C09087=1078.769,309.066,-90.171,175.453,27.389,154.727
C09088=1078.775,309.314,-90.203,175.457,27.393,154.728
C09089=1078.781,309.562,-90.235,175.459,27.397,154.729
C09090=1078.787,309.810,-90.267,175.462,27.402,154.729
C09091=1078.793,310.058,-90.299,175.465,27.406,154.730
C09092=1078.799,310.305,-90.330,175.468,27.410,154.730
C09093=1078.805,310.553,-90.362,175.471,27.415,154.731
C09094=1078.811,310.801,-90.394,175.474,27.419,154.732
C09095=1078.817,311.049,-90.426,175.477,27.423,154.733
C09096=1078.823,311.297,-90.458,175.480,27.427,154.733
C09097=1078.829,311.545,-90.490,175.483,27.432,154.734
C09098=1078.835,311.793,-90.522,175.486,27.436,154.735
C09099=1078.841,312.040,-90.553,175.489,27.440,154.735
C09100=1078.847,312.289,-90.585,175.492,27.444,154.736
C09101=1078.853,312.536,-90.618,175.495,27.448,154.736
C09102=1078.859,312.783,-90.649,175.497,27.452,154.737
C09103=1078.865,313.032,-90.681,175.501,27.457,154.738
C09104=1078.871,313.280,-90.713,175.504,27.461,154.738
C09105=1078.877,313.527,-90.746,175.507,27.465,154.739
C09106=1078.883,313.776,-90.778,175.510,27.469,154.740
C09107=1078.889,314.023,-90.810,175.512,27.474,154.740
C09108=1078.895,314.271,-90.841,175.515,27.478,154.741
C09109=1078.902,314.519,-90.874,175.519,27.482,154.742
C09110=1078.908,314.767,-90.906,175.522,27.487,154.742
C09111=1078.914,315.015,-90.938,175.525,27.491,154.743
C09112=1078.919,315.262,-90.971,175.527,27.495,154.744
C09113=1078.925,315.511,-91.003,175.530,27.500,154.745
C09114=1078.931,315.758,-91.036,175.534,27.504,154.745
C09115=1078.936,316.006,-91.067,175.537,27.509,154.746
C09116=1078.942,316.254,-91.101,175.539,27.513,154.747
C09117=1078.947,316.467,-91.129,175.542,27.517,154.747
C09118=1078.952,316.679,-91.156,175.544,27.521,154.748
C09119=1078.957,316.892,-91.184,175.547,27.524,154.748
C09120=1078.962,317.104,-91.212,175.550,27.528,154.749
C09121=1078.967,317.317,-91.240,175.552,27.532,154.750
C09122=1078.972,317.530,-91.268,175.555,27.536,154.750
C09123=1078.977,317.742,-91.295,175.557,27.540,154.751
C09124=1078.982,317.955,-91.323,175.560,27.543,154.751
C09125=1078.988,318.203,-91.355,175.562,27.548,154.752
C09126=1078.993,318.451,-91.388,175.566,27.552,154.753
C09127=1078.999,318.699,-91.420,175.569,27.557,154.754
C09128=1079.005,318.946,-91.453,175.572,27.561,154.754
C09129=1079.011,319.194,-91.486,175.575,27.566,154.755
C09130=1079.017,319.443,-91.518,175.578,27.570,154.756
C09131=1079.023,319.690,-91.551,175.580,27.575,154.757
C09132=1079.028,319.937,-91.584,175.583,27.579,154.757
C09133=1079.034,320.186,-91.616,175.587,27.584,154.758
C09134=1079.041,320.433,-91.649,175.590,27.588,154.759
C09135=1079.046,320.681,-91.682,175.593,27.593,154.759
C09136=1079.052,320.929,-91.715,175.596,27.597,154.760
C09137=1079.058,321.177,-91.747,175.598,27.601,154.761
C09138=1079.064,321.425,-91.780,175.602,27.606,154.762
C09139=1079.070,321.672,-91.813,175.605,27.611,154.762
C09140=1079.077,321.920,-91.846,175.608,27.615,154.763
C09141=1079.082,322.168,-91.879,175.611,27.620,154.764
C09142=1079.087,322.415,-91.911,175.614,27.624,154.764
C09143=1079.093,322.663,-91.944,175.617,27.629,154.765
C09144=1079.099,322.911,-91.977,175.619,27.633,154.766
C09145=1079.106,323.158,-92.010,175.623,27.637,154.767
C09146=1079.111,323.406,-92.043,175.626,27.642,154.767
C09147=1079.117,323.654,-92.076,175.629,27.647,154.768
C09148=1079.123,323.902,-92.109,175.632,27.651,154.769
C09149=1079.129,324.149,-92.142,175.635,27.656,154.770
C09150=1079.135,324.397,-92.175,175.638,27.661,154.770
C09151=1079.141,324.645,-92.208,175.642,27.665,154.771
C09152=1079.147,324.893,-92.241,175.644,27.669,154.772
C09153=1079.153,325.140,-92.274,175.647,27.674,154.773
C09154=1079.160,325.389,-92.307,175.650,27.678,154.773
C09155=1079.165,325.637,-92.340,175.653,27.683,154.774
C09156=1079.172,325.884,-92.373,175.656,27.688,154.775
C09157=1079.177,326.132,-92.407,175.660,27.692,154.775
C09158=1079.184,326.380,-92.439,175.663,27.697,154.776
C09159=1079.189,326.628,-92.473,175.666,27.701,154.777
C09160=1079.195,326.875,-92.505,175.669,27.706,154.778
C09161=1079.201,327.123,-92.539,175.672,27.710,154.778
C09162=1079.208,327.370,-92.572,175.675,27.715,154.779
C09163=1079.213,327.618,-92.605,175.678,27.720,154.780
C09164=1079.220,327.866,-92.639,175.681,27.724,154.781
C09165=1079.226,328.114,-92.672,175.684,27.728,154.781
C09166=1079.232,328.361,-92.705,175.687,27.733,154.782
C09167=1079.238,328.609,-92.739,175.690,27.738,154.783
C09168=1079.244,328.857,-92.771,175.693,27.743,154.784
C09169=1079.250,329.105,-92.805,175.697,27.747,154.785
C09170=1079.257,329.352,-92.839,175.700,27.752,154.785
C09171=1079.262,329.600,-92.872,175.703,27.756,154.786
C09172=1079.269,329.848,-92.905,175.706,27.761,154.787
C09173=1079.279,330.266,-92.961,175.712,27.769,154.788
C09174=1079.289,330.685,-93.018,175.716,27.776,154.789
C09175=1079.300,331.104,-93.075,175.722,27.785,154.791
C09176=1079.310,331.523,-93.131,175.727,27.793,154.792
C09177=1079.316,331.770,-93.165,175.731,27.797,154.793
C09178=1079.322,332.018,-93.199,175.734,27.802,154.793
C09179=1079.328,332.266,-93.232,175.737,27.807,154.794
C09180=1079.334,332.513,-93.266,175.740,27.812,154.795
C09181=1079.340,332.761,-93.299,175.743,27.816,154.796
C09182=1079.346,333.009,-93.333,175.746,27.821,154.797
C09183=1079.352,333.257,-93.367,175.749,27.826,154.797
C09184=1079.358,333.504,-93.401,175.753,27.831,154.798
C09185=1079.364,333.752,-93.435,175.756,27.836,154.799
C09186=1079.369,334.000,-93.468,175.759,27.840,154.800
C09187=1079.376,334.247,-93.502,175.762,27.845,154.801
C09188=1079.382,334.495,-93.536,175.765,27.850,154.801
C09189=1079.388,334.742,-93.570,175.768,27.855,154.802
C09190=1079.394,334.990,-93.604,175.771,27.860,154.803
C09191=1079.400,335.238,-93.638,175.775,27.864,154.804
C09192=1079.406,335.486,-93.671,175.778,27.870,154.805
C09193=1079.411,335.733,-93.706,175.781,27.874,154.805
C09194=1079.418,335.981,-93.740,175.784,27.879,154.806
C09195=1079.424,336.228,-93.774,175.787,27.884,154.807
C09196=1079.430,336.475,-93.808,175.790,27.889,154.808
C09197=1079.436,336.724,-93.842,175.793,27.894,154.809
C09198=1079.442,336.971,-93.876,175.797,27.898,154.809
C09199=1079.448,337.219,-93.910,175.800,27.904,154.810
C09200=1079.455,337.466,-93.944,175.803,27.908,154.811
C09201=1079.461,337.714,-93.978,175.806,27.913,154.812
C09202=1079.467,337.962,-94.012,175.809,27.918,154.813
C09203=1079.473,338.209,-94.046,175.812,27.923,154.814
C09204=1079.478,338.456,-94.081,175.815,27.928,154.815
C09205=1079.484,338.704,-94.115,175.819,27.933,154.815
C09206=1079.490,338.952,-94.149,175.822,27.938,154.816
C09207=1079.496,339.199,-94.183,175.825,27.943,154.817
C09208=1079.503,339.447,-94.218,175.828,27.948,154.818
C09209=1079.509,339.694,-94.252,175.831,27.952,154.819
C09210=1079.515,339.942,-94.286,175.834,27.958,154.820
C09211=1079.520,340.190,-94.321,175.837,27.963,154.820
C09212=1079.526,340.437,-94.355,175.840,27.968,154.821
C09213=1079.532,340.685,-94.389,175.844,27.973,154.822
C09214=1079.538,340.932,-94.423,175.848,27.978,154.823
C09215=1079.545,341.180,-94.458,175.851,27.983,154.824
C09216=1079.551,341.428,-94.492,175.854,27.988,154.825
C09217=1079.556,341.676,-94.527,175.857,27.993,154.825
C09218=1079.563,341.923,-94.562,175.860,27.998,154.826
C09219=1079.569,342.171,-94.596,175.863,28.003,154.827
C09220=1079.575,342.418,-94.630,175.866,28.008,154.828
C09221=1079.581,342.666,-94.665,175.870,28.013,154.829
C09222=1079.587,342.913,-94.700,175.873,28.018,154.830
C09223=1079.593,343.161,-94.734,175.876,28.023,154.831
C09224=1079.599,343.408,-94.768,175.879,28.028,154.832
C09225=1079.609,343.822,-94.827,175.884,28.037,154.833
C09226=1079.619,344.235,-94.884,175.890,28.045,154.834
C09227=1079.630,344.648,-94.942,175.895,28.054,154.836
C09228=1079.640,345.061,-95.000,175.901,28.062,154.837
C09229=1079.646,345.309,-95.035,175.904,28.067,154.838
C09230=1079.651,345.556,-95.070,175.907,28.073,154.839
C09231=1079.658,345.804,-95.105,175.910,28.078,154.840
C09232=1079.664,346.052,-95.140,175.914,28.083,154.841
C09233=1079.670,346.299,-95.174,175.918,28.088,154.842
C09234=1079.676,346.547,-95.210,175.921,28.094,154.843
C09235=1079.682,346.794,-95.244,175.924,28.099,154.844
C09236=1079.688,347.042,-95.279,175.927,28.104,154.845
C09237=1079.694,347.289,-95.315,175.930,28.109,154.846
C09238=1079.700,347.537,-95.349,175.933,28.114,154.846
C09239=1079.706,347.784,-95.385,175.937,28.120,154.847
C09240=1079.712,348.032,-95.419,175.940,28.125,154.848
C09241=1079.718,348.279,-95.455,175.943,28.131,154.849
C09242=1079.725,348.527,-95.490,175.946,28.136,154.850
C09243=1079.730,348.774,-95.525,175.950,28.141,154.851
C09244=1079.737,349.022,-95.559,175.953,28.146,154.852
C09245=1079.743,349.269,-95.595,175.957,28.152,154.853
C09246=1079.748,349.516,-95.631,175.960,28.157,154.854
C09247=1079.755,349.764,-95.666,175.963,28.162,154.855
C09248=1079.761,350.012,-95.701,175.966,28.168,154.856
C09249=1079.767,350.258,-95.735,175.969,28.173,154.857
C09250=1079.773,350.506,-95.771,175.973,28.179,154.858
C09251=1079.780,350.754,-95.806,175.976,28.184,154.859
C09252=1079.785,351.001,-95.842,175.979,28.189,154.859
C09253=1079.791,351.248,-95.877,175.983,28.195,154.860
C09254=1079.798,351.496,-95.912,175.986,28.200,154.861
C09255=1079.804,351.744,-95.948,175.990,28.205,154.862
C09256=1079.810,351.991,-95.982,175.993,28.211,154.863
C09257=1079.816,352.238,-96.018,175.996,28.216,154.864
C09258=1079.822,352.486,-96.054,175.999,28.221,154.865
C09259=1079.829,352.733,-96.089,176.002,28.227,154.866
C09260=1079.834,352.980,-96.124,176.006,28.232,154.867
C09261=1079.840,353.228,-96.160,176.009,28.238,154.868
C09262=1079.847,353.475,-96.195,176.012,28.243,154.869
C09263=1079.853,353.723,-96.231,176.016,28.249,154.870
C09264=1079.859,353.969,-96.267,176.020,28.254,154.871
C09265=1079.865,354.217,-96.303,176.023,28.260,154.872
C09266=1079.871,354.465,-96.338,176.026,28.265,154.873
C09267=1079.878,354.712,-96.374,176.029,28.271,154.874
C09268=1079.884,354.960,-96.409,176.033,28.276,154.875
C09269=1079.889,355.207,-96.445,176.036,28.282,154.876
C09270=1079.895,355.454,-96.481,176.039,28.287,154.877
C09271=1079.901,355.701,-96.517,176.042,28.293,154.878
C09272=1079.907,355.949,-96.553,176.046,28.299,154.879
C09273=1079.914,356.196,-96.588,176.049,28.304,154.880
C09274=1079.921,356.443,-96.624,176.052,28.310,154.881
C09275=1079.926,356.690,-96.660,176.056,28.315,154.882
C09276=1079.932,356.938,-96.695,176.060,28.321,154.883
C09277=1079.941,357.295,-96.747,176.064,28.329,154.884
C09278=1079.950,357.652,-96.799,176.069,28.337,154.886
C09279=1079.959,358.010,-96.851,176.074,28.345,154.887
C09280=1079.968,358.367,-96.903,176.078,28.353,154.889
C09281=1079.974,358.615,-96.939,176.082,28.359,154.890
C09282=1079.981,358.862,-96.975,176.085,28.365,154.891
C09283=1079.987,359.110,-97.011,176.089,28.371,154.892
C09284=1079.993,359.357,-97.047,176.093,28.377,154.893
C09285=1079.999,359.603,-97.083,176.096,28.382,154.894
C09286=1080.005,359.851,-97.119,176.099,28.388,154.895
C09287=1080.011,360.098,-97.156,176.103,28.394,154.896
C09288=1080.017,360.345,-97.191,176.106,28.399,154.897
C09289=1080.023,360.592,-97.228,176.109,28.405,154.898
C09290=1080.030,360.839,-97.264,176.113,28.411,154.899
C09291=1080.036,361.087,-97.300,176.116,28.417,154.900
C09292=1080.042,361.334,-97.336,176.119,28.423,154.901
C09293=1080.050,361.641,-97.381,176.124,28.430,154.902
C09294=1080.057,361.948,-97.426,176.128,28.437,154.904
C09295=1080.065,362.254,-97.471,176.132,28.444,154.905
C09296=1080.072,362.560,-97.517,176.136,28.452,154.906
C09297=1080.079,362.807,-97.553,176.140,28.457,154.907
C09298=1080.085,363.055,-97.589,176.144,28.463,154.908
C09299=1080.091,363.302,-97.625,176.147,28.469,154.910
C09300=1080.098,363.550,-97.662,176.150,28.475,154.911
C09301=1080.104,363.797,-97.699,176.154,28.481,154.912
C09302=1080.111,364.044,-97.735,176.157,28.487,154.913
C09303=1080.116,364.291,-97.772,176.160,28.493,154.914
C09304=1080.123,364.538,-97.809,176.164,28.499,154.915
C09305=1080.129,364.785,-97.845,176.167,28.505,154.916
C09306=1080.135,365.032,-97.881,176.171,28.511,154.917
C09307=1080.142,365.280,-97.918,176.174,28.517,154.918
C09308=1080.147,365.527,-97.955,176.177,28.523,154.919
C09309=1080.154,365.774,-97.991,176.181,28.529,154.921
C09310=1080.160,366.021,-98.028,176.184,28.535,154.922
C09311=1080.166,366.268,-98.065,176.188,28.541,154.923
C09312=1080.173,366.516,-98.102,176.191,28.547,154.924
C09313=1080.178,366.764,-98.139,176.194,28.553,154.925
C09314=1080.184,367.011,-98.175,176.198,28.560,154.926
C09315=1080.191,367.258,-98.212,176.201,28.566,154.927
C09316=1080.197,367.504,-98.249,176.206,28.572,154.928
C09317=1080.203,367.751,-98.286,176.209,28.578,154.930
C09318=1080.209,367.999,-98.323,176.212,28.584,154.931
C09319=1080.216,368.247,-98.360,176.216,28.590,154.932
C09320=1080.222,368.494,-98.396,176.219,28.596,154.933
C09321=1080.228,368.740,-98.434,176.223,28.603,154.934
C09322=1080.234,368.987,-98.470,176.226,28.609,154.935
C09323=1080.240,369.235,-98.507,176.230,28.615,154.936
C09324=1080.247,369.482,-98.545,176.233,28.621,154.938
C09325=1080.253,369.729,-98.582,176.237,28.627,154.939
C09326=1080.259,369.976,-98.619,176.240,28.633,154.940
C09327=1080.265,370.223,-98.656,176.243,28.640,154.941
C09328=1080.271,370.470,-98.693,176.247,28.646,154.942
C09329=1080.277,370.687,-98.726,176.250,28.651,154.943
C09330=1080.283,370.903,-98.758,176.253,28.657,154.944
C09331=1080.288,371.119,-98.791,176.257,28.663,154.945
C09332=1080.294,371.335,-98.823,176.260,28.668,154.946
C09333=1080.299,371.551,-98.856,176.262,28.674,154.947
C09334=1080.305,371.768,-98.889,176.265,28.679,154.949
C09335=1080.310,371.985,-98.921,176.268,28.685,154.950
C09336=1080.315,372.201,-98.953,176.271,28.690,154.951
C09337=1080.323,372.448,-98.991,176.275,28.697,154.952
C09338=1080.328,372.695,-99.029,176.278,28.703,154.953
C09339=1080.335,372.942,-99.065,176.282,28.710,154.954
C09340=1080.341,373.189,-99.103,176.285,28.716,154.955
C09341=1080.348,373.436,-99.140,176.290,28.722,154.956
C09342=1080.354,373.684,-99.178,176.293,28.728,154.958
C09343=1080.360,373.931,-99.215,176.297,28.735,154.959
C09344=1080.367,374.177,-99.253,176.300,28.741,154.960
C09345=1080.372,374.424,-99.290,176.304,28.748,154.961
C09346=1080.379,374.672,-99.328,176.307,28.754,154.963
C09347=1080.385,374.919,-99.366,176.311,28.761,154.964
C09348=1080.391,375.166,-99.404,176.314,28.768,154.965
C09349=1080.398,375.412,-99.441,176.318,28.774,154.966
C09350=1080.404,375.659,-99.479,176.321,28.781,154.968
C09351=1080.410,375.907,-99.517,176.325,28.787,154.969
C09352=1080.416,376.154,-99.554,176.329,28.794,154.970
C09353=1080.423,376.400,-99.591,176.332,28.801,154.972
C09354=1080.429,376.648,-99.629,176.336,28.808,154.973
C09355=1080.435,376.895,-99.667,176.339,28.814,154.974
C09356=1080.441,377.142,-99.705,176.343,28.820,154.975
C09357=1080.447,377.389,-99.743,176.346,28.827,154.977
C09358=1080.454,377.636,-99.781,176.350,28.834,154.978
C09359=1080.461,377.882,-99.819,176.353,28.840,154.979
C09360=1080.467,378.129,-99.856,176.357,28.847,154.980
C09361=1080.473,378.376,-99.895,176.361,28.854,154.982
C09362=1080.479,378.623,-99.932,176.364,28.861,154.983
C09363=1080.486,378.870,-99.970,176.368,28.868,154.984
C09364=1080.492,379.117,-100.008,176.371,28.874,154.986
C09365=1080.498,379.365,-100.046,176.375,28.881,154.987
C09366=1080.505,379.610,-100.084,176.379,28.888,154.988
C09367=1080.511,379.858,-100.122,176.382,28.894,154.989
C09368=1080.518,380.105,-100.160,176.386,28.902,154.991
C09369=1080.524,380.352,-100.198,176.389,28.908,154.992
C09370=1080.531,380.599,-100.237,176.393,28.915,154.993
C09371=1080.537,380.846,-100.275,176.397,28.922,154.995
C09372=1080.543,381.093,-100.313,176.400,28.929,154.996
C09373=1080.549,381.339,-100.351,176.404,28.936,154.997
C09374=1080.556,381.587,-100.389,176.408,28.943,154.999
C09375=1080.563,381.834,-100.428,176.411,28.950,155.000
C09376=1080.569,382.080,-100.465,176.415,28.956,155.001
C09377=1080.575,382.328,-100.504,176.419,28.964,155.003
C09378=1080.581,382.574,-100.543,176.422,28.971,155.004
C09379=1080.588,382.821,-100.581,176.426,28.978,155.006
C09380=1080.595,383.068,-100.620,176.430,28.985,155.007
C09381=1080.601,383.314,-100.658,176.433,28.992,155.008
C09382=1080.607,383.562,-100.696,176.437,28.999,155.010
C09383=1080.613,383.808,-100.735,176.441,29.006,155.011
C09384=1080.619,384.056,-100.773,176.444,29.013,155.013
C09385=1080.625,384.286,-100.810,176.448,29.020,155.014
C09386=1080.632,384.517,-100.845,176.451,29.027,155.015
C09387=1080.638,384.747,-100.881,176.454,29.033,155.016
C09388=1080.644,384.978,-100.918,176.458,29.040,155.018
C09389=1080.650,385.209,-100.954,176.461,29.047,155.019
C09390=1080.656,385.439,-100.990,176.465,29.054,155.020
C09391=1080.661,385.670,-101.026,176.468,29.060,155.022
C09392=1080.667,385.900,-101.063,176.472,29.067,155.023
C09393=1080.674,386.147,-101.101,176.475,29.074,155.024
C09394=1080.680,386.393,-101.140,176.479,29.082,155.026
C09395=1080.686,386.641,-101.179,176.483,29.089,155.027
C09396=1080.693,386.888,-101.217,176.486,29.096,155.029
C09397=1080.699,387.134,-101.256,176.490,29.103,155.030
C09398=1080.706,387.381,-101.295,176.494,29.111,155.032
C09399=1080.712,387.628,-101.334,176.498,29.118,155.033
C09400=1080.719,387.875,-101.373,176.501,29.125,155.034
C09401=1080.725,388.121,-101.411,176.505,29.133,155.036
C09402=1080.732,388.368,-101.450,176.509,29.140,155.037
C09403=1080.738,388.615,-101.490,176.513,29.148,155.039
C09404=1080.745,388.862,-101.529,176.516,29.155,155.040
C09405=1080.752,389.109,-101.567,176.520,29.163,155.042
C09406=1080.758,389.356,-101.607,176.524,29.170,155.043
C09407=1080.764,389.601,-101.646,176.528,29.178,155.045
C09408=1080.771,389.848,-101.685,176.532,29.185,155.046
C09409=1080.777,390.095,-101.724,176.535,29.192,155.048
C09410=1080.784,390.342,-101.763,176.539,29.200,155.049
C09411=1080.791,390.589,-101.802,176.543,29.207,155.051
C09412=1080.797,390.835,-101.842,176.547,29.215,155.052
C09413=1080.804,391.082,-101.881,176.551,29.223,155.054
C09414=1080.811,391.329,-101.920,176.554,29.230,155.055
C09415=1080.817,391.576,-101.959,176.558,29.238,155.057
C09416=1080.824,391.822,-101.999,176.562,29.246,155.058
C09417=1080.830,392.070,-102.038,176.566,29.253,155.060
C09418=1080.837,392.316,-102.077,176.570,29.261,155.061
C09419=1080.843,392.563,-102.117,176.574,29.269,155.063
C09420=1080.849,392.810,-102.157,176.577,29.276,155.065
C09421=1080.856,393.056,-102.196,176.581,29.284,155.066
C09422=1080.862,393.303,-102.236,176.585,29.292,155.068
C09423=1080.870,393.550,-102.275,176.589,29.300,155.069
C09424=1080.876,393.797,-102.315,176.593,29.308,155.071
C09425=1080.882,394.043,-102.355,176.597,29.315,155.072
C09426=1080.889,394.290,-102.394,176.601,29.323,155.074
C09427=1080.895,394.537,-102.434,176.604,29.331,155.076
C09428=1080.902,394.783,-102.473,176.608,29.339,155.077
C09429=1080.908,395.030,-102.513,176.612,29.347,155.079
C09430=1080.915,395.276,-102.553,176.616,29.355,155.080
C09431=1080.921,395.523,-102.592,176.620,29.363,155.082
C09432=1080.928,395.770,-102.632,176.624,29.371,155.084
C09433=1080.934,396.016,-102.672,176.628,29.379,155.085
C09434=1080.941,396.263,-102.712,176.632,29.387,155.087
C09435=1080.947,396.510,-102.752,176.636,29.395,155.089
C09436=1080.954,396.757,-102.792,176.639,29.403,155.090
C09437=1080.961,397.003,-102.832,176.643,29.411,155.092
C09438=1080.967,397.250,-102.872,176.647,29.419,155.093
C09439=1080.974,397.496,-102.912,176.651,29.427,155.095
C09440=1080.980,397.743,-102.951,176.655,29.436,155.097
C09441=1080.986,397.981,-102.990,176.659,29.444,155.098
C09442=1080.993,398.219,-103.029,176.663,29.451,155.100
C09443=1080.999,398.456,-103.068,176.666,29.459,155.102
C09444=1081.006,398.694,-103.106,176.670,29.467,155.103
C09445=1081.012,398.931,-103.145,176.674,29.475,155.105
C09446=1081.019,399.170,-103.184,176.678,29.483,155.107
C09447=1081.025,399.407,-103.223,176.682,29.491,155.108
C09448=1081.031,399.645,-103.261,176.685,29.499,155.110
C09449=1081.037,399.892,-103.301,176.689,29.508,155.112
C09450=1081.044,400.139,-103.342,176.692,29.516,155.113
C09451=1081.051,400.386,-103.382,176.696,29.524,155.115
C09452=1081.057,400.632,-103.423,176.700,29.533,155.117
C09453=1081.064,400.878,-103.463,176.704,29.541,155.118
C09454=1081.071,401.125,-103.504,176.708,29.550,155.120
C09455=1081.077,401.372,-103.544,176.712,29.558,155.122
C09456=1081.083,401.618,-103.584,176.716,29.567,155.124
C09457=1081.091,401.865,-103.625,176.720,29.575,155.125
C09458=1081.097,402.111,-103.665,176.725,29.584,155.127
C09459=1081.104,402.359,-103.706,176.729,29.593,155.129
C09460=1081.111,402.604,-103.747,176.733,29.601,155.131
C09461=1081.117,402.851,-103.787,176.737,29.610,155.133
C09462=1081.124,403.098,-103.828,176.741,29.619,155.134
C09463=1081.131,403.344,-103.868,176.745,29.627,155.136
C09464=1081.138,403.591,-103.909,176.749,29.636,155.138
C09465=1081.144,403.838,-103.950,176.753,29.644,155.140
C09466=1081.151,404.085,-103.991,176.757,29.653,155.142
C09467=1081.157,404.331,-104.031,176.761,29.662,155.143
C09468=1081.164,404.577,-104.072,176.765,29.671,155.145
C09469=1081.171,404.824,-104.113,176.769,29.679,155.147
C09470=1081.177,405.070,-104.154,176.774,29.689,155.149
C09471=1081.184,405.317,-104.195,176.778,29.697,155.151
C09472=1081.191,405.563,-104.236,176.782,29.706,155.153
C09473=1081.197,405.810,-104.278,176.786,29.716,155.155
C09474=1081.204,406.056,-104.318,176.790,29.724,155.156
C09475=1081.211,406.303,-104.359,176.794,29.733,155.158
C09476=1081.218,406.549,-104.400,176.797,29.742,155.160
C09477=1081.224,406.796,-104.442,176.802,29.752,155.162
C09478=1081.231,407.043,-104.482,176.806,29.760,155.164
C09479=1081.238,407.289,-104.523,176.810,29.769,155.166
C09480=1081.244,407.536,-104.565,176.814,29.778,155.168
C09481=1081.251,407.782,-104.606,176.818,29.788,155.170
C09482=1081.258,408.029,-104.647,176.823,29.797,155.172
C09483=1081.265,408.275,-104.689,176.827,29.806,155.174
C09484=1081.271,408.521,-104.730,176.831,29.815,155.176
C09485=1081.278,408.768,-104.771,176.835,29.825,155.177
C09486=1081.284,409.014,-104.813,176.839,29.834,155.180
C09487=1081.291,409.261,-104.854,176.844,29.843,155.181
C09488=1081.298,409.508,-104.896,176.848,29.853,155.183
C09489=1081.305,409.754,-104.937,176.852,29.862,155.185
C09490=1081.311,410.001,-104.979,176.856,29.872,155.187
C09491=1081.318,410.247,-105.020,176.861,29.881,155.189
C09492=1081.325,410.493,-105.062,176.865,29.890,155.191
C09493=1081.331,410.740,-105.104,176.869,29.900,155.193
C09494=1081.339,410.986,-105.145,176.874,29.909,155.195
C09495=1081.345,411.233,-105.187,176.878,29.919,155.197
C09496=1081.352,411.478,-105.228,176.882,29.928,155.199
C09497=1081.359,411.718,-105.269,176.886,29.937,155.201
C09498=1081.366,411.957,-105.309,176.891,29.947,155.203
C09499=1081.372,412.196,-105.350,176.895,29.956,155.205
C09500=1081.379,412.434,-105.390,176.899,29.966,155.207
C09501=1081.385,412.673,-105.430,176.903,29.975,155.209
C09502=1081.392,412.912,-105.472,176.907,29.984,155.211
C09503=1081.399,413.150,-105.512,176.912,29.994,155.213
C09504=1081.405,413.390,-105.553,176.916,30.004,155.215
C09505=1081.413,413.636,-105.595,176.920,30.013,155.217
C09506=1081.419,413.882,-105.636,176.925,30.023,155.219
C09507=1081.426,414.128,-105.679,176.928,30.033,155.222
C09508=1081.433,414.374,-105.721,176.932,30.042,155.224
C09509=1081.440,414.621,-105.762,176.937,30.053,155.226
C09510=1081.447,414.867,-105.805,176.941,30.062,155.228
C09511=1081.454,415.113,-105.847,176.946,30.072,155.230
C09512=1081.461,415.360,-105.889,176.950,30.082,155.232
C09513=1081.468,415.606,-105.931,176.955,30.092,155.234
C09514=1081.475,415.853,-105.974,176.959,30.102,155.236
C09515=1081.482,416.099,-106.016,176.964,30.112,155.239
C09516=1081.489,416.346,-106.057,176.968,30.123,155.241
C09517=1081.496,416.592,-106.100,176.972,30.133,155.243
C09518=1081.502,416.838,-106.143,176.977,30.143,155.245
C09519=1081.509,417.084,-106.185,176.981,30.153,155.247
C09520=1081.516,417.331,-106.228,176.986,30.164,155.250
C09521=1081.523,417.577,-106.270,176.991,30.174,155.252
C09522=1081.530,417.823,-106.313,176.995,30.184,155.254
C09523=1081.537,418.070,-106.355,177.000,30.194,155.256
C09524=1081.543,418.316,-106.398,177.004,30.205,155.259
C09525=1081.550,418.562,-106.440,177.009,30.215,155.261
C09526=1081.558,418.808,-106.484,177.013,30.226,155.263
C09527=1081.564,419.054,-106.526,177.018,30.236,155.265
C09528=1081.571,419.300,-106.569,177.022,30.247,155.268
C09529=1081.578,419.547,-106.611,177.027,30.257,155.270
C09530=1081.585,419.793,-106.654,177.032,30.268,155.272
C09531=1081.592,420.039,-106.697,177.036,30.278,155.275
C09532=1081.599,420.285,-106.740,177.041,30.289,155.277
C09533=1081.606,420.532,-106.782,177.045,30.300,155.279
C09534=1081.614,420.778,-106.826,177.050,30.310,155.282
C09535=1081.620,421.024,-106.868,177.055,30.321,155.284
C09536=1081.628,421.270,-106.912,177.059,30.331,155.286
C09537=1081.634,421.516,-106.954,177.064,30.342,155.289
C09538=1081.642,421.762,-106.998,177.069,30.353,155.291
C09539=1081.649,422.008,-107.040,177.073,30.364,155.293
C09540=1081.655,422.254,-107.084,177.078,30.375,155.296
C09541=1081.662,422.501,-107.127,177.083,30.386,155.298
C09542=1081.670,422.747,-107.170,177.088,30.397,155.300
C09543=1081.677,422.993,-107.213,177.092,30.408,155.303
C09544=1081.683,423.239,-107.257,177.097,30.419,155.305
C09545=1081.691,423.485,-107.300,177.102,30.430,155.308
C09546=1081.698,423.731,-107.343,177.106,30.441,155.310
C09547=1081.705,423.977,-107.387,177.111,30.452,155.313
C09548=1081.712,424.224,-107.430,177.116,30.464,155.315
C09549=1081.719,424.469,-107.473,177.121,30.475,155.318
C09550=1081.727,424.716,-107.517,177.125,30.486,155.320
C09551=1081.733,424.962,-107.561,177.130,30.497,155.323
C09552=1081.740,425.207,-107.604,177.135,30.509,155.325
C09553=1081.747,425.455,-107.648,177.140,30.520,155.327
C09554=1081.755,425.703,-107.692,177.145,30.531,155.330
C09555=1081.762,425.951,-107.735,177.150,30.543,155.333
C09556=1081.769,426.200,-107.780,177.155,30.554,155.335
C09557=1081.776,426.446,-107.824,177.159,30.566,155.338
C09558=1081.784,426.692,-107.867,177.164,30.577,155.340
C09559=1081.790,426.937,-107.911,177.169,30.589,155.343
C09560=1081.798,427.183,-107.955,177.174,30.600,155.345
C09561=1081.805,427.429,-107.998,177.179,30.612,155.348
C09562=1081.812,427.676,-108.042,177.184,30.624,155.351
C09563=1081.820,427.921,-108.086,177.189,30.636,155.353
C09564=1081.827,428.167,-108.131,177.194,30.647,155.356
C09565=1081.834,428.413,-108.174,177.198,30.659,155.358
C09566=1081.841,428.659,-108.219,177.203,30.671,155.361
C09567=1081.848,428.905,-108.262,177.208,30.682,155.364
C09568=1081.856,429.151,-108.307,177.213,30.694,155.366
C09569=1081.862,429.397,-108.351,177.218,30.706,155.369
C09570=1081.870,429.643,-108.395,177.223,30.718,155.372
C09571=1081.877,429.889,-108.439,177.228,30.731,155.374
C09572=1081.885,430.134,-108.483,177.234,30.742,155.377
C09573=1081.892,430.381,-108.528,177.239,30.755,155.380
C09574=1081.898,430.626,-108.572,177.244,30.767,155.383
C09575=1081.907,430.872,-108.616,177.249,30.779,155.385
C09576=1081.914,431.119,-108.661,177.254,30.791,155.388
C09577=1081.920,431.364,-108.705,177.259,30.803,155.391
C09578=1081.928,431.610,-108.750,177.264,30.816,155.394
C09579=1081.936,431.856,-108.795,177.269,30.828,155.396
C09580=1081.942,432.101,-108.839,177.274,30.841,155.399
C09581=1081.950,432.347,-108.883,177.279,30.853,155.402
C09582=1081.958,432.594,-108.928,177.284,30.865,155.405
C09583=1081.965,432.840,-108.973,177.290,30.878,155.408
C09584=1081.972,433.085,-109.017,177.295,30.891,155.410
C09585=1081.979,433.331,-109.062,177.300,30.903,155.413
C09586=1081.987,433.577,-109.108,177.306,30.916,155.416
C09587=1081.993,433.822,-109.152,177.311,30.929,155.419
C09588=1082.001,434.068,-109.197,177.316,30.941,155.422
C09589=1082.008,434.314,-109.242,177.321,30.954,155.425
C09590=1082.016,434.560,-109.287,177.326,30.967,155.428
C09591=1082.023,434.806,-109.331,177.332,30.980,155.431
C09592=1082.030,435.051,-109.377,177.337,30.993,155.434
C09593=1082.038,435.297,-109.422,177.342,31.006,155.436
C09594=1082.045,435.543,-109.467,177.347,31.019,155.439
C09595=1082.053,435.788,-109.512,177.353,31.032,155.442
C09596=1082.060,436.034,-109.557,177.359,31.045,155.445
C09597=1082.068,436.280,-109.603,177.364,31.058,155.448
C09598=1082.075,436.526,-109.648,177.369,31.071,155.451
C09599=1082.083,436.771,-109.693,177.374,31.084,155.454
C09600=1082.090,437.017,-109.738,177.380,31.098,155.457
C09601=1082.097,437.262,-109.784,177.385,31.111,155.461
C09602=1082.105,437.507,-109.829,177.391,31.124,155.463
C09603=1082.112,437.753,-109.874,177.396,31.137,155.467
C09604=1082.120,438.000,-109.920,177.402,31.151,155.470
C09605=1082.128,438.245,-109.966,177.407,31.165,155.473
C09606=1082.135,438.491,-110.011,177.412,31.178,155.476
C09607=1082.143,438.736,-110.056,177.418,31.191,155.479
C09608=1082.150,438.982,-110.102,177.424,31.205,155.482
C09609=1082.159,439.265,-110.155,177.430,31.221,155.486
C09610=1082.167,439.548,-110.207,177.437,31.236,155.489
C09611=1082.176,439.831,-110.260,177.443,31.252,155.493
C09612=1082.185,440.114,-110.313,177.450,31.268,155.497
C09613=1082.193,440.361,-110.359,177.455,31.282,155.500
C09614=1082.200,440.606,-110.405,177.460,31.296,155.503
C09615=1082.207,440.852,-110.451,177.466,31.310,155.506
C09616=1082.215,441.097,-110.497,177.472,31.324,155.510
C09617=1082.223,441.342,-110.543,177.478,31.339,155.513
C09618=1082.230,441.588,-110.589,177.483,31.352,155.516
C09619=1082.238,441.834,-110.635,177.489,31.367,155.519
C09620=1082.246,442.079,-110.681,177.495,31.381,155.523
C09621=1082.253,442.324,-110.728,177.501,31.396,155.526
C09622=1082.261,442.570,-110.774,177.506,31.410,155.529
C09623=1082.268,442.816,-110.821,177.512,31.424,155.533
C09624=1082.276,443.061,-110.867,177.518,31.438,155.536
C09625=1082.284,443.306,-110.913,177.524,31.453,155.539
C09626=1082.291,443.552,-110.959,177.529,31.467,155.543
C09627=1082.299,443.797,-111.006,177.535,31.482,155.546
C09628=1082.306,444.043,-111.052,177.542,31.497,155.550
C09629=1082.315,444.288,-111.099,177.547,31.511,155.553
C09630=1082.322,444.534,-111.146,177.553,31.526,155.557
C09631=1082.330,444.778,-111.192,177.559,31.541,155.560
C09632=1082.338,445.025,-111.239,177.565,31.556,155.564
C09633=1082.345,445.270,-111.285,177.571,31.571,155.567
C09634=1082.353,445.515,-111.333,177.576,31.586,155.571
C09635=1082.361,445.760,-111.379,177.583,31.601,155.574
C09636=1082.369,446.006,-111.426,177.588,31.616,155.578
C09637=1082.376,446.251,-111.473,177.593,31.631,155.581
C09638=1082.385,446.497,-111.520,177.599,31.646,155.585
C09639=1082.392,446.742,-111.567,177.603,31.660,155.588
C09640=1082.400,446.988,-111.614,177.608,31.675,155.592
C09641=1082.408,447.232,-111.661,177.612,31.690,155.596
C09642=1082.416,447.478,-111.708,177.616,31.705,155.599
C09643=1082.423,447.723,-111.756,177.621,31.720,155.603
C09644=1082.432,447.968,-111.802,177.624,31.735,155.606
C09645=1082.439,448.214,-111.850,177.628,31.750,155.610
C09646=1082.447,448.459,-111.897,177.631,31.765,155.614
C09647=1082.455,448.704,-111.945,177.635,31.780,155.617
C09648=1082.463,448.950,-111.991,177.637,31.795,155.621
C09649=1082.471,449.194,-112.039,177.640,31.809,155.625
C09650=1082.479,449.439,-112.085,177.642,31.824,155.628
C09651=1082.490,449.685,-112.131,177.646,31.837,155.632
C09652=1082.503,449.931,-112.176,177.648,31.850,155.635
C09653=1082.134,449.923,-112.391,177.618,32.024,155.681
C09654=1082.121,449.678,-112.346,177.616,32.011,155.678
C09655=1082.110,449.432,-112.301,177.613,31.998,155.675
C09656=1082.102,449.187,-112.254,177.610,31.983,155.671
C09657=1082.094,448.942,-112.207,177.608,31.969,155.667
C09658=1082.086,448.697,-112.159,177.604,31.954,155.664
C09659=1082.077,448.452,-112.112,177.601,31.939,155.660
C09660=1082.070,448.206,-112.065,177.597,31.924,155.656
C09661=1082.062,447.961,-112.017,177.593,31.909,155.653
C09662=1082.053,447.716,-111.970,177.590,31.894,155.649
C09663=1082.046,447.471,-111.923,177.585,31.879,155.645
C09664=1082.038,447.225,-111.876,177.582,31.864,155.642
C09665=1082.030,446.981,-111.829,177.577,31.849,155.638
C09666=1082.022,446.735,-111.782,177.572,31.834,155.635
C09667=1082.014,446.489,-111.734,177.567,31.819,155.631
C09668=1082.006,446.244,-111.688,177.562,31.805,155.628
C09669=1081.998,445.998,-111.641,177.556,31.789,155.624
C09670=1081.991,445.753,-111.594,177.551,31.774,155.620
C09671=1081.983,445.508,-111.547,177.545,31.760,155.617
C09672=1081.975,445.263,-111.500,177.539,31.744,155.613
C09673=1081.968,445.017,-111.453,177.533,31.730,155.610
C09674=1081.960,444.772,-111.406,177.526,31.715,155.606
C09675=1081.952,444.526,-111.359,177.521,31.700,155.603
C09676=1081.944,444.281,-111.313,177.515,31.685,155.599
C09677=1081.937,444.036,-111.266,177.508,31.670,155.596
C09678=1081.928,443.790,-111.220,177.503,31.656,155.592
C09679=1081.921,443.545,-111.173,177.496,31.641,155.589
C09680=1081.913,443.299,-111.127,177.491,31.627,155.586
C09681=1081.905,443.054,-111.080,177.485,31.612,155.582
C09682=1081.898,442.808,-111.034,177.479,31.598,155.579
C09683=1081.890,442.563,-110.987,177.473,31.583,155.576
C09684=1081.883,442.317,-110.941,177.468,31.569,155.572
C09685=1081.875,442.072,-110.895,177.461,31.555,155.569
C09686=1081.867,441.827,-110.849,177.456,31.540,155.566
C09687=1081.859,441.581,-110.802,177.450,31.526,155.562
C09688=1081.852,441.336,-110.756,177.444,31.512,155.559
C09689=1081.844,441.090,-110.710,177.438,31.498,155.556
C09690=1081.837,440.844,-110.664,177.433,31.484,155.552
C09691=1081.829,440.599,-110.617,177.426,31.470,155.549
C09692=1081.821,440.353,-110.572,177.421,31.456,155.546
C09693=1081.814,440.108,-110.525,177.415,31.442,155.543
C09694=1081.805,439.840,-110.475,177.409,31.427,155.539
C09695=1081.798,439.573,-110.426,177.403,31.412,155.536
C09696=1081.789,439.305,-110.376,177.397,31.397,155.532
C09697=1081.780,439.039,-110.326,177.391,31.382,155.529
C09698=1081.773,438.793,-110.280,177.385,31.368,155.526
C09699=1081.766,438.548,-110.235,177.379,31.355,155.523
C09700=1081.758,438.301,-110.189,177.374,31.341,155.519
C09701=1081.750,438.055,-110.144,177.368,31.328,155.516
C09702=1081.743,437.810,-110.098,177.363,31.314,155.513
C09703=1081.735,437.564,-110.052,177.357,31.301,155.510
C09704=1081.727,437.319,-110.007,177.351,31.287,155.507
C09705=1081.720,437.073,-109.962,177.346,31.274,155.504
C09706=1081.712,436.828,-109.916,177.341,31.261,155.501
C09707=1081.705,436.582,-109.870,177.335,31.248,155.498
C09708=1081.697,436.336,-109.826,177.329,31.234,155.495
C09709=1081.690,436.091,-109.780,177.324,31.221,155.492
C09710=1081.682,435.845,-109.735,177.319,31.209,155.489
C09711=1081.675,435.600,-109.690,177.313,31.195,155.486
C09712=1081.668,435.354,-109.645,177.308,31.182,155.483
C09713=1081.661,435.108,-109.600,177.302,31.169,155.480
C09714=1081.653,434.862,-109.554,177.297,31.156,155.477
C09715=1081.646,434.616,-109.509,177.292,31.144,155.474
C09716=1081.638,434.370,-109.464,177.286,31.131,155.471
C09717=1081.630,434.125,-109.419,177.281,31.118,155.468
C09718=1081.623,433.880,-109.375,177.276,31.105,155.466
C09719=1081.616,433.634,-109.330,177.271,31.092,155.463
C09720=1081.609,433.388,-109.285,177.265,31.080,155.460
C09721=1081.601,433.142,-109.240,177.260,31.067,155.457
C09722=1081.595,432.896,-109.195,177.254,31.054,155.454
C09723=1081.587,432.650,-109.150,177.249,31.042,155.451
C09724=1081.580,432.405,-109.105,177.244,31.030,155.448
C09725=1081.573,432.158,-109.061,177.239,31.017,155.446
C09726=1081.565,431.913,-109.017,177.234,31.005,155.443
C09727=1081.558,431.667,-108.972,177.229,30.992,155.440
C09728=1081.550,431.421,-108.927,177.223,30.980,155.437
C09729=1081.542,431.175,-108.882,177.218,30.968,155.434
C09730=1081.536,430.930,-108.838,177.213,30.955,155.432
C09731=1081.528,430.684,-108.793,177.208,30.943,155.429
C09732=1081.521,430.437,-108.749,177.203,30.931,155.426
C09733=1081.514,430.192,-108.705,177.198,30.919,155.423
C09734=1081.507,429.946,-108.660,177.193,30.907,155.421
C09735=1081.499,429.700,-108.616,177.187,30.895,155.418
C09736=1081.492,429.454,-108.572,177.182,30.883,155.415
C09737=1081.484,429.208,-108.528,177.177,30.871,155.413
C09738=1081.478,428.963,-108.483,177.172,30.859,155.410
C09739=1081.470,428.716,-108.439,177.167,30.847,155.407
C09740=1081.463,428.471,-108.395,177.162,30.835,155.405
C09741=1081.456,428.224,-108.351,177.157,30.823,155.402
C09742=1081.449,427.979,-108.307,177.152,30.811,155.399
C09743=1081.442,427.732,-108.263,177.147,30.800,155.397
C09744=1081.434,427.487,-108.220,177.142,30.788,155.394
C09745=1081.426,427.241,-108.175,177.137,30.777,155.392
C09746=1081.420,426.995,-108.131,177.132,30.765,155.389
C09747=1081.412,426.749,-108.088,177.127,30.753,155.386
C09748=1081.406,426.503,-108.044,177.122,30.741,155.384
C09749=1081.398,426.257,-108.000,177.117,30.730,155.381
C09750=1081.391,426.007,-107.955,177.112,30.718,155.379
C09751=1081.383,425.759,-107.911,177.108,30.707,155.376
C09752=1081.376,425.509,-107.867,177.103,30.695,155.374
C09753=1081.369,425.259,-107.823,177.097,30.684,155.371
C09754=1081.362,425.014,-107.780,177.092,30.673,155.369
C09755=1081.354,424.767,-107.736,177.087,30.661,155.366
C09756=1081.348,424.521,-107.692,177.083,30.650,155.364
C09757=1081.340,424.275,-107.649,177.078,30.639,155.361
C09758=1081.333,424.029,-107.605,177.073,30.628,155.359
C09759=1081.326,423.783,-107.561,177.068,30.616,155.356
C09760=1081.319,423.538,-107.518,177.064,30.605,155.354
C09761=1081.311,423.291,-107.475,177.059,30.594,155.351
C09762=1081.305,423.045,-107.431,177.054,30.583,155.349
C09763=1081.298,422.799,-107.388,177.049,30.572,155.346
C09764=1081.290,422.553,-107.345,177.045,30.561,155.344
C09765=1081.284,422.306,-107.302,177.040,30.550,155.342
C09766=1081.277,422.060,-107.258,177.035,30.539,155.339
C09767=1081.270,421.815,-107.215,177.030,30.529,155.337
C09768=1081.263,421.568,-107.172,177.025,30.517,155.334
C09769=1081.255,421.322,-107.129,177.020,30.507,155.332
C09770=1081.248,421.076,-107.086,177.016,30.496,155.330
C09771=1081.241,420.830,-107.043,177.011,30.485,155.327
C09772=1081.234,420.583,-107.000,177.006,30.475,155.325
C09773=1081.227,420.337,-106.957,177.002,30.464,155.323
C09774=1081.220,420.091,-106.914,176.997,30.453,155.320
C09775=1081.213,419.845,-106.872,176.993,30.443,155.318
C09776=1081.206,419.599,-106.829,176.988,30.432,155.316
C09777=1081.199,419.353,-106.786,176.983,30.421,155.313
C09778=1081.192,419.107,-106.743,176.979,30.411,155.311
C09779=1081.185,418.860,-106.701,176.974,30.401,155.309
C09780=1081.178,418.614,-106.657,176.970,30.390,155.307
C09781=1081.171,418.368,-106.615,176.965,30.380,155.304
C09782=1081.164,418.121,-106.572,176.961,30.369,155.302
C09783=1081.157,417.875,-106.530,176.956,30.359,155.300
C09784=1081.150,417.629,-106.487,176.952,30.349,155.298
C09785=1081.143,417.382,-106.445,176.946,30.338,155.295
C09786=1081.136,417.136,-106.402,176.942,30.328,155.293
C09787=1081.130,416.890,-106.359,176.937,30.318,155.291
C09788=1081.123,416.644,-106.317,176.933,30.308,155.289
C09789=1081.116,416.397,-106.274,176.928,30.297,155.287
C09790=1081.109,416.151,-106.232,176.924,30.287,155.284
C09791=1081.102,415.905,-106.189,176.919,30.277,155.282
C09792=1081.095,415.658,-106.147,176.915,30.267,155.280
C09793=1081.088,415.413,-106.105,176.910,30.257,155.278
C09794=1081.081,415.166,-106.063,176.906,30.247,155.276
C09795=1081.074,414.919,-106.020,176.901,30.237,155.274
C09796=1081.067,414.673,-105.979,176.897,30.227,155.271
C09797=1081.060,414.426,-105.937,176.893,30.217,155.269
C09798=1081.053,414.180,-105.894,176.888,30.207,155.267
C09799=1081.046,413.934,-105.852,176.884,30.197,155.265
C09800=1081.039,413.687,-105.810,176.879,30.188,155.263
C09801=1081.033,413.442,-105.768,176.875,30.178,155.261
C09802=1081.025,413.202,-105.728,176.871,30.169,155.259
C09803=1081.019,412.963,-105.687,176.867,30.159,155.257
C09804=1081.012,412.723,-105.646,176.862,30.149,155.255
C09805=1081.005,412.484,-105.605,176.858,30.140,155.253
C09806=1080.999,412.245,-105.565,176.854,30.131,155.251
C09807=1080.992,412.005,-105.524,176.850,30.121,155.249
C09808=1080.985,411.766,-105.483,176.846,30.112,155.247
C09809=1080.979,411.526,-105.443,176.841,30.102,155.245
C09810=1080.972,411.280,-105.401,176.836,30.093,155.243
C09811=1080.965,411.033,-105.360,176.832,30.083,155.241
C09812=1080.958,410.786,-105.318,176.828,30.074,155.239
C09813=1080.952,410.541,-105.276,176.823,30.065,155.237
C09814=1080.944,410.294,-105.234,176.819,30.055,155.235
C09815=1080.938,410.047,-105.193,176.815,30.045,155.233
C09816=1080.931,409.801,-105.152,176.810,30.036,155.231
C09817=1080.925,409.554,-105.110,176.806,30.027,155.229
C09818=1080.917,409.308,-105.068,176.802,30.018,155.227
C09819=1080.911,409.062,-105.027,176.798,30.008,155.225
C09820=1080.904,408.816,-104.985,176.794,29.999,155.223
C09821=1080.897,408.569,-104.943,176.789,29.990,155.221
C09822=1080.891,408.323,-104.903,176.785,29.980,155.219
C09823=1080.884,408.076,-104.861,176.781,29.971,155.217
C09824=1080.877,407.829,-104.820,176.777,29.962,155.215
C09825=1080.871,407.583,-104.778,176.773,29.953,155.213
C09826=1080.864,407.337,-104.737,176.768,29.943,155.211
C09827=1080.858,407.090,-104.695,176.764,29.934,155.209
C09828=1080.851,406.843,-104.655,176.760,29.925,155.207
C09829=1080.843,406.597,-104.614,176.756,29.916,155.205
C09830=1080.837,406.350,-104.572,176.752,29.907,155.204
C09831=1080.830,406.104,-104.531,176.748,29.898,155.202
C09832=1080.823,405.858,-104.490,176.743,29.889,155.200
C09833=1080.817,405.610,-104.449,176.739,29.880,155.198
C09834=1080.810,405.364,-104.408,176.735,29.871,155.196
C09835=1080.803,405.118,-104.367,176.731,29.862,155.194
C09836=1080.797,404.871,-104.327,176.727,29.854,155.192
C09837=1080.790,404.624,-104.285,176.723,29.844,155.190
C09838=1080.784,404.379,-104.244,176.719,29.836,155.189
C09839=1080.777,404.131,-104.204,176.715,29.827,155.187
C09840=1080.770,403.885,-104.163,176.711,29.818,155.185
C09841=1080.763,403.638,-104.122,176.707,29.810,155.183
C09842=1080.756,403.392,-104.081,176.702,29.801,155.181
C09843=1080.750,403.145,-104.040,176.698,29.792,155.180
C09844=1080.743,402.899,-103.999,176.694,29.783,155.178
C09845=1080.736,402.652,-103.959,176.690,29.775,155.176
C09846=1080.730,402.406,-103.918,176.686,29.766,155.174
C09847=1080.723,402.159,-103.878,176.682,29.758,155.172
C09848=1080.716,401.912,-103.837,176.678,29.749,155.171
C09849=1080.710,401.666,-103.796,176.674,29.740,155.169
C09850=1080.703,401.419,-103.756,176.670,29.732,155.167
C09851=1080.696,401.172,-103.716,176.666,29.723,155.165
C09852=1080.690,400.926,-103.676,176.662,29.715,155.164
C09853=1080.683,400.679,-103.634,176.658,29.706,155.162
C09854=1080.676,400.433,-103.594,176.654,29.698,155.160
C09855=1080.670,400.186,-103.554,176.650,29.690,155.158
C09856=1080.663,399.940,-103.514,176.646,29.681,155.157
C09857=1080.656,399.693,-103.473,176.642,29.673,155.155
C09858=1080.650,399.454,-103.434,176.638,29.665,155.153
C09859=1080.644,399.216,-103.395,176.635,29.657,155.152
C09860=1080.637,398.978,-103.357,176.631,29.649,155.150
C09861=1080.631,398.739,-103.318,176.627,29.640,155.148
C09862=1080.625,398.500,-103.279,176.622,29.632,155.147
C09863=1080.618,398.263,-103.240,176.618,29.625,155.145
C09864=1080.612,398.024,-103.201,176.615,29.617,155.143
C09865=1080.605,397.786,-103.162,176.611,29.609,155.142
C09866=1080.599,397.539,-103.122,176.607,29.600,155.140
C09867=1080.592,397.293,-103.082,176.603,29.592,155.138
C09868=1080.586,397.046,-103.042,176.599,29.584,155.137
C09869=1080.580,396.799,-103.002,176.595,29.576,155.135
C09870=1080.572,396.552,-102.963,176.591,29.568,155.133
C09871=1080.566,396.306,-102.922,176.588,29.560,155.132
C09872=1080.559,396.059,-102.882,176.584,29.552,155.130
C09873=1080.553,395.813,-102.842,176.580,29.544,155.129
C09874=1080.546,395.566,-102.803,176.576,29.536,155.127
C09875=1080.540,395.319,-102.763,176.572,29.528,155.125
C09876=1080.533,395.073,-102.723,176.568,29.520,155.124
C09877=1080.527,394.826,-102.684,176.564,29.512,155.122
C09878=1080.520,394.580,-102.644,176.560,29.504,155.120
C09879=1080.513,394.332,-102.604,176.557,29.496,155.119
C09880=1080.507,394.085,-102.564,176.553,29.488,155.117
C09881=1080.500,393.839,-102.525,176.549,29.480,155.116
C09882=1080.494,393.592,-102.485,176.545,29.473,155.114
C09883=1080.487,393.345,-102.445,176.541,29.464,155.112
C09884=1080.481,393.099,-102.406,176.537,29.457,155.111
C09885=1080.474,392.852,-102.366,176.533,29.449,155.109
C09886=1080.467,392.605,-102.327,176.530,29.442,155.108
C09887=1080.461,392.359,-102.287,176.526,29.433,155.106
C09888=1080.454,392.112,-102.248,176.522,29.426,155.105
C09889=1080.448,391.865,-102.208,176.518,29.418,155.103
C09890=1080.442,391.618,-102.169,176.514,29.410,155.102
C09891=1080.435,391.371,-102.130,176.511,29.403,155.100
C09892=1080.428,391.125,-102.090,176.507,29.395,155.098
C09893=1080.422,390.878,-102.051,176.503,29.387,155.097
C09894=1080.415,390.631,-102.012,176.499,29.380,155.096
C09895=1080.408,390.386,-101.973,176.495,29.372,155.094
C09896=1080.402,390.139,-101.933,176.492,29.365,155.092
C09897=1080.396,389.892,-101.894,176.488,29.357,155.091
C09898=1080.389,389.645,-101.856,176.484,29.350,155.089
C09899=1080.383,389.398,-101.816,176.480,29.342,155.088
C09900=1080.376,389.151,-101.777,176.476,29.335,155.086
C09901=1080.369,388.905,-101.738,176.472,29.328,155.085
C09902=1080.363,388.658,-101.698,176.468,29.320,155.083
C09903=1080.356,388.411,-101.660,176.464,29.313,155.082
C09904=1080.350,388.165,-101.621,176.460,29.305,155.081
C09905=1080.344,387.918,-101.582,176.457,29.298,155.079
C09906=1080.337,387.671,-101.543,176.453,29.290,155.078
C09907=1080.330,387.424,-101.504,176.449,29.283,155.076
C09908=1080.323,387.177,-101.465,176.445,29.276,155.075
C09909=1080.318,386.931,-101.426,176.442,29.268,155.073
C09910=1080.311,386.684,-101.387,176.438,29.261,155.072
C09911=1080.304,386.437,-101.348,176.434,29.254,155.070
C09912=1080.298,386.190,-101.310,176.430,29.247,155.069
C09913=1080.292,385.943,-101.271,176.427,29.239,155.067
C09914=1080.286,385.712,-101.235,176.423,29.232,155.066
C09915=1080.280,385.481,-101.198,176.420,29.226,155.065
C09916=1080.273,385.249,-101.162,176.417,29.219,155.063
C09917=1080.267,385.018,-101.126,176.413,29.212,155.062
C09918=1080.261,384.787,-101.090,176.410,29.206,155.061
C09919=1080.256,384.555,-101.054,176.406,29.198,155.060
C09920=1080.250,384.324,-101.017,176.402,29.192,155.058
C09921=1080.244,384.093,-100.981,176.399,29.185,155.057
C09922=1080.237,383.846,-100.943,176.395,29.178,155.056
C09923=1080.231,383.600,-100.904,176.391,29.171,155.054
C09924=1080.224,383.353,-100.865,176.388,29.164,155.053
C09925=1080.218,383.106,-100.828,176.384,29.157,155.051
C09926=1080.212,382.859,-100.788,176.380,29.149,155.050
C09927=1080.206,382.612,-100.750,176.377,29.143,155.049
C09928=1080.199,382.366,-100.712,176.373,29.135,155.047
C09929=1080.193,382.118,-100.673,176.369,29.128,155.046
C09930=1080.187,381.872,-100.635,176.366,29.122,155.044
C09931=1080.180,381.625,-100.597,176.362,29.114,155.043
C09932=1080.173,381.378,-100.558,176.359,29.108,155.042
C09933=1080.167,381.131,-100.520,176.355,29.101,155.040
C09934=1080.161,380.884,-100.481,176.351,29.094,155.039
C09935=1080.154,380.637,-100.443,176.348,29.087,155.038
C09936=1080.148,380.390,-100.406,176.344,29.080,155.036
C09937=1080.141,380.143,-100.367,176.341,29.074,155.035
C09938=1080.135,379.897,-100.330,176.337,29.066,155.034
C09939=1080.128,379.649,-100.291,176.332,29.059,155.032
C09940=1080.122,379.402,-100.253,176.329,29.053,155.031
C09941=1080.116,379.156,-100.215,176.325,29.046,155.030
C09942=1080.109,378.908,-100.177,176.322,29.039,155.028
C09943=1080.103,378.662,-100.139,176.318,29.032,155.027
C09944=1080.097,378.414,-100.101,176.314,29.026,155.026
C09945=1080.091,378.167,-100.063,176.311,29.019,155.025
C09946=1080.084,377.920,-100.026,176.307,29.012,155.023
C09947=1080.077,377.674,-99.987,176.304,29.006,155.022
C09948=1080.071,377.427,-99.949,176.300,28.999,155.021
C09949=1080.065,377.180,-99.911,176.297,28.992,155.020
C09950=1080.059,376.933,-99.873,176.293,28.986,155.018
C09951=1080.052,376.686,-99.835,176.289,28.979,155.017
C09952=1080.046,376.439,-99.798,176.286,28.972,155.016
C09953=1080.039,376.192,-99.760,176.282,28.965,155.014
C09954=1080.033,375.945,-99.722,176.279,28.959,155.013
C09955=1080.027,375.698,-99.684,176.275,28.952,155.012
C09956=1080.021,375.451,-99.646,176.272,28.945,155.011
C09957=1080.015,375.204,-99.610,176.267,28.939,155.009
C09958=1080.008,374.956,-99.572,176.264,28.933,155.008
C09959=1080.002,374.710,-99.534,176.260,28.926,155.007
C09960=1079.996,374.463,-99.496,176.257,28.919,155.006
C09961=1079.989,374.216,-99.459,176.253,28.913,155.004
C09962=1079.983,373.969,-99.421,176.250,28.906,155.003
C09963=1079.978,373.722,-99.384,176.246,28.900,155.002
C09964=1079.970,373.475,-99.346,176.243,28.894,155.001
C09965=1079.964,373.228,-99.309,176.239,28.887,154.999
C09966=1079.958,372.980,-99.271,176.236,28.881,154.998
C09967=1079.952,372.733,-99.234,176.232,28.874,154.997
C09968=1079.946,372.487,-99.196,176.229,28.868,154.996
C09969=1079.939,372.239,-99.160,176.225,28.861,154.995
C09970=1079.934,372.022,-99.127,176.221,28.856,154.994
C09971=1079.928,371.805,-99.094,176.218,28.850,154.993
C09972=1079.923,371.588,-99.061,176.216,28.845,154.991
C09973=1079.917,371.371,-99.028,176.213,28.839,154.990
C09974=1079.911,371.155,-98.996,176.210,28.834,154.989
C09975=1079.906,370.938,-98.963,176.207,28.828,154.988
C09976=1079.900,370.720,-98.931,176.203,28.823,154.987
C09977=1079.895,370.504,-98.898,176.200,28.817,154.986
C09978=1079.888,370.257,-98.860,176.197,28.811,154.985
C09979=1079.882,370.009,-98.823,176.193,28.804,154.984
C09980=1079.875,369.763,-98.786,176.190,28.798,154.983
C09981=1079.870,369.516,-98.749,176.186,28.792,154.982
C09982=1079.863,369.268,-98.712,176.183,28.786,154.980
C09983=1079.857,369.021,-98.675,176.179,28.779,154.979
C09984=1079.851,368.774,-98.638,176.176,28.773,154.978
C09985=1079.844,368.527,-98.602,176.173,28.767,154.977
C09986=1079.838,368.280,-98.564,176.169,28.761,154.976
C09987=1079.832,368.033,-98.527,176.165,28.755,154.975
C09988=1079.826,367.785,-98.490,176.161,28.749,154.973
C09989=1079.819,367.539,-98.453,176.158,28.742,154.972
C09990=1079.813,367.292,-98.417,176.154,28.736,154.971
C09991=1079.807,367.044,-98.379,176.151,28.730,154.970
C09992=1079.801,366.797,-98.343,176.148,28.724,154.969
C09993=1079.795,366.550,-98.306,176.144,28.718,154.968
C09994=1079.788,366.302,-98.269,176.141,28.712,154.967
C09995=1079.782,366.056,-98.232,176.138,28.706,154.965
C09996=1079.776,365.808,-98.195,176.134,28.700,154.964
//INST
///DATE 2021/06/17 10:54
///ATTR SC,RW,RJ
////FRAME ROBOT
///GROUP1 RB1
NOP
MOVL C00000 V=800.0 PL=0
MOVL C00001 V=800.0 PL=0
MOVL C00002 V=800.0 PL=0
MOVL C00003 V=800.0 PL=0
MOVL C00004 V=800.0 PL=0
MOVL C00005 V=800.0 PL=0
MOVL C00006 V=800.0 PL=0
MOVL C00007 V=800.0 PL=0
MOVL C00008 V=800.0 PL=0
MOVL C00009 V=800.0 PL=0
MOVL C00010 V=800.0 PL=0
MOVL C00011 V=800.0 PL=0
MOVL C00012 V=800.0 PL=0
MOVL C00013 V=800.0 PL=0
MOVL C00014 V=800.0 PL=0
MOVL C00015 V=800.0 PL=0
MOVL C00016 V=800.0 PL=0
MOVL C00017 V=800.0 PL=0
MOVL C00018 V=800.0 PL=0
MOVL C00019 V=800.0 PL=0
MOVL C00020 V=800.0 PL=0
MOVL C00021 V=800.0 PL=0
MOVL C00022 V=800.0 PL=0
MOVL C00023 V=800.0 PL=0
MOVL C00024 V=800.0 PL=0
MOVL C00025 V=800.0 PL=0
MOVL C00026 V=800.0 PL=0
MOVL C00027 V=800.0 PL=0
MOVL C00028 V=800.0 PL=0
MOVL C00029 V=800.0 PL=0
MOVL C00030 V=800.0 PL=0
MOVL C00031 V=800.0 PL=0
MOVL C00032 V=800.0 PL=0
MOVL C00033 V=800.0 PL=0
MOVL C00034 V=800.0 PL=0
MOVL C00035 V=800.0 PL=0
MOVL C00036 V=800.0 PL=0
MOVL C00037 V=800.0 PL=0
MOVL C00038 V=800.0 PL=0
MOVL C00039 V=800.0 PL=0
MOVL C00040 V=800.0 PL=0
MOVL C00041 V=800.0 PL=0
MOVL C00042 V=800.0 PL=0
MOVL C00043 V=800.0 PL=0
MOVL C00044 V=800.0 PL=0
MOVL C00045 V=800.0 PL=0
MOVL C00046 V=800.0 PL=0
MOVL C00047 V=800.0 PL=0
MOVL C00048 V=800.0 PL=0
MOVL C00049 V=800.0 PL=0
MOVL C00050 V=800.0 PL=0
MOVL C00051 V=800.0 PL=0
MOVL C00052 V=800.0 PL=0
MOVL C00053 V=800.0 PL=0
MOVL C00054 V=800.0 PL=0
MOVL C00055 V=800.0 PL=0
MOVL C00056 V=800.0 PL=0
MOVL C00057 V=800.0 PL=0
MOVL C00058 V=800.0 PL=0
MOVL C00059 V=800.0 PL=0
MOVL C00060 V=800.0 PL=0
MOVL C00061 V=800.0 PL=0
MOVL C00062 V=800.0 PL=0
MOVL C00063 V=800.0 PL=0
MOVL C00064 V=800.0 PL=0
MOVL C00065 V=800.0 PL=0
MOVL C00066 V=800.0 PL=0
MOVL C00067 V=800.0 PL=0
MOVL C00068 V=800.0 PL=0
MOVL C00069 V=800.0 PL=0
MOVL C00070 V=800.0 PL=0
MOVL C00071 V=800.0 PL=0
MOVL C00072 V=800.0 PL=0
MOVL C00073 V=800.0 PL=0
MOVL C00074 V=800.0 PL=0
MOVL C00075 V=800.0 PL=0
MOVL C00076 V=800.0 PL=0
MOVL C00077 V=800.0 PL=0
MOVL C00078 V=800.0 PL=0
MOVL C00079 V=800.0 PL=0
MOVL C00080 V=800.0 PL=0
MOVL C00081 V=800.0 PL=0
MOVL C00082 V=800.0 PL=0
MOVL C00083 V=800.0 PL=0
MOVL C00084 V=800.0 PL=0
MOVL C00085 V=800.0 PL=0
MOVL C00086 V=800.0 PL=0
MOVL C00087 V=800.0 PL=0
MOVL C00088 V=800.0 PL=0
MOVL C00089 V=800.0 PL=0
MOVL C00090 V=800.0 PL=0
MOVL C00091 V=800.0 PL=0
MOVL C00092 V=800.0 PL=0
MOVL C00093 V=800.0 PL=0
MOVL C00094 V=800.0 PL=0
MOVL C00095 V=800.0 PL=0
MOVL C00096 V=800.0 PL=0
MOVL C00097 V=800.0 PL=0
MOVL C00098 V=800.0 PL=0
MOVL C00099 V=800.0 PL=0
MOVL C00100 V=800.0 PL=0
MOVL C00101 V=800.0 PL=0
MOVL C00102 V=800.0 PL=0
MOVL C00103 V=800.0 PL=0
MOVL C00104 V=800.0 PL=0
MOVL C00105 V=800.0 PL=0
MOVL C00106 V=800.0 PL=0
MOVL C00107 V=800.0 PL=0
MOVL C00108 V=800.0 PL=0
MOVL C00109 V=800.0 PL=0
MOVL C00110 V=800.0 PL=0
MOVL C00111 V=800.0 PL=0
MOVL C00112 V=800.0 PL=0
MOVL C00113 V=800.0 PL=0
MOVL C00114 V=800.0 PL=0
MOVL C00115 V=800.0 PL=0
MOVL C00116 V=800.0 PL=0
MOVL C00117 V=800.0 PL=0
MOVL C00118 V=800.0 PL=0
MOVL C00119 V=800.0 PL=0
MOVL C00120 V=800.0 PL=0
MOVL C00121 V=800.0 PL=0
MOVL C00122 V=800.0 PL=0
MOVL C00123 V=800.0 PL=0
MOVL C00124 V=800.0 PL=0
MOVL C00125 V=800.0 PL=0
MOVL C00126 V=800.0 PL=0
MOVL C00127 V=800.0 PL=0
MOVL C00128 V=800.0 PL=0
MOVL C00129 V=800.0 PL=0
MOVL C00130 V=800.0 PL=0
MOVL C00131 V=800.0 PL=0
MOVL C00132 V=800.0 PL=0
MOVL C00133 V=800.0 PL=0
MOVL C00134 V=800.0 PL=0
MOVL C00135 V=800.0 PL=0
MOVL C00136 V=800.0 PL=0
MOVL C00137 V=800.0 PL=0
MOVL C00138 V=800.0 PL=0
MOVL C00139 V=800.0 PL=0
MOVL C00140 V=800.0 PL=0
MOVL C00141 V=800.0 PL=0
MOVL C00142 V=800.0 PL=0
MOVL C00143 V=800.0 PL=0
MOVL C00144 V=800.0 PL=0
MOVL C00145 V=800.0 PL=0
MOVL C00146 V=800.0 PL=0
MOVL C00147 V=800.0 PL=0
MOVL C00148 V=800.0 PL=0
MOVL C00149 V=800.0 PL=0
MOVL C00150 V=800.0 PL=0
MOVL C00151 V=800.0 PL=0
MOVL C00152 V=800.0 PL=0
MOVL C00153 V=800.0 PL=0
MOVL C00154 V=800.0 PL=0
MOVL C00155 V=800.0 PL=0
MOVL C00156 V=800.0 PL=0
MOVL C00157 V=800.0 PL=0
MOVL C00158 V=800.0 PL=0
MOVL C00159 V=800.0 PL=0
MOVL C00160 V=800.0 PL=0
MOVL C00161 V=800.0 PL=0
MOVL C00162 V=800.0 PL=0
MOVL C00163 V=800.0 PL=0
MOVL C00164 V=800.0 PL=0
MOVL C00165 V=800.0 PL=0
MOVL C00166 V=800.0 PL=0
MOVL C00167 V=800.0 PL=0
MOVL C00168 V=800.0 PL=0
MOVL C00169 V=800.0 PL=0
MOVL C00170 V=800.0 PL=0
MOVL C00171 V=800.0 PL=0
MOVL C00172 V=800.0 PL=0
MOVL C00173 V=800.0 PL=0
MOVL C00174 V=800.0 PL=0
MOVL C00175 V=800.0 PL=0
MOVL C00176 V=800.0 PL=0
MOVL C00177 V=800.0 PL=0
MOVL C00178 V=800.0 PL=0
MOVL C00179 V=800.0 PL=0
MOVL C00180 V=800.0 PL=0
MOVL C00181 V=800.0 PL=0
MOVL C00182 V=800.0 PL=0
MOVL C00183 V=800.0 PL=0
MOVL C00184 V=800.0 PL=0
MOVL C00185 V=800.0 PL=0
MOVL C00186 V=800.0 PL=0
MOVL C00187 V=800.0 PL=0
MOVL C00188 V=800.0 PL=0
MOVL C00189 V=800.0 PL=0
MOVL C00190 V=800.0 PL=0
MOVL C00191 V=800.0 PL=0
MOVL C00192 V=800.0 PL=0
MOVL C00193 V=800.0 PL=0
MOVL C00194 V=800.0 PL=0
MOVL C00195 V=800.0 PL=0
MOVL C00196 V=800.0 PL=0
MOVL C00197 V=800.0 PL=0
MOVL C00198 V=800.0 PL=0
MOVL C00199 V=800.0 PL=0
MOVL C00200 V=800.0 PL=0
MOVL C00201 V=800.0 PL=0
MOVL C00202 V=800.0 PL=0
MOVL C00203 V=800.0 PL=0
MOVL C00204 V=800.0 PL=0
MOVL C00205 V=800.0 PL=0
MOVL C00206 V=800.0 PL=0
MOVL C00207 V=800.0 PL=0
MOVL C00208 V=800.0 PL=0
MOVL C00209 V=800.0 PL=0
MOVL C00210 V=800.0 PL=0
MOVL C00211 V=800.0 PL=0
MOVL C00212 V=800.0 PL=0
MOVL C00213 V=800.0 PL=0
MOVL C00214 V=800.0 PL=0
MOVL C00215 V=800.0 PL=0
MOVL C00216 V=800.0 PL=0
MOVL C00217 V=800.0 PL=0
MOVL C00218 V=800.0 PL=0
MOVL C00219 V=800.0 PL=0
MOVL C00220 V=800.0 PL=0
MOVL C00221 V=800.0 PL=0
MOVL C00222 V=800.0 PL=0
MOVL C00223 V=800.0 PL=0
MOVL C00224 V=800.0 PL=0
MOVL C00225 V=800.0 PL=0
MOVL C00226 V=800.0 PL=0
MOVL C00227 V=800.0 PL=0
MOVL C00228 V=800.0 PL=0
MOVL C00229 V=800.0 PL=0
MOVL C00230 V=800.0 PL=0
MOVL C00231 V=800.0 PL=0
MOVL C00232 V=800.0 PL=0
MOVL C00233 V=800.0 PL=0
MOVL C00234 V=800.0 PL=0
MOVL C00235 V=800.0 PL=0
MOVL C00236 V=800.0 PL=0
MOVL C00237 V=800.0 PL=0
MOVL C00238 V=800.0 PL=0
MOVL C00239 V=800.0 PL=0
MOVL C00240 V=800.0 PL=0
MOVL C00241 V=800.0 PL=0
MOVL C00242 V=800.0 PL=0
MOVL C00243 V=800.0 PL=0
MOVL C00244 V=800.0 PL=0
MOVL C00245 V=800.0 PL=0
MOVL C00246 V=800.0 PL=0
MOVL C00247 V=800.0 PL=0
MOVL C00248 V=800.0 PL=0
MOVL C00249 V=800.0 PL=0
MOVL C00250 V=800.0 PL=0
MOVL C00251 V=800.0 PL=0
MOVL C00252 V=800.0 PL=0
MOVL C00253 V=800.0 PL=0
MOVL C00254 V=800.0 PL=0
MOVL C00255 V=800.0 PL=0
MOVL C00256 V=800.0 PL=0
MOVL C00257 V=800.0 PL=0
MOVL C00258 V=800.0 PL=0
MOVL C00259 V=800.0 PL=0
MOVL C00260 V=800.0 PL=0
MOVL C00261 V=800.0 PL=0
MOVL C00262 V=800.0 PL=0
MOVL C00263 V=800.0 PL=0
MOVL C00264 V=800.0 PL=0
MOVL C00265 V=800.0 PL=0
MOVL C00266 V=800.0 PL=0
MOVL C00267 V=800.0 PL=0
MOVL C00268 V=800.0 PL=0
MOVL C00269 V=800.0 PL=0
MOVL C00270 V=800.0 PL=0
MOVL C00271 V=800.0 PL=0
MOVL C00272 V=800.0 PL=0
MOVL C00273 V=800.0 PL=0
MOVL C00274 V=800.0 PL=0
MOVL C00275 V=800.0 PL=0
MOVL C00276 V=800.0 PL=0
MOVL C00277 V=800.0 PL=0
MOVL C00278 V=800.0 PL=0
MOVL C00279 V=800.0 PL=0
MOVL C00280 V=800.0 PL=0
MOVL C00281 V=800.0 PL=0
MOVL C00282 V=800.0 PL=0
MOVL C00283 V=800.0 PL=0
MOVL C00284 V=800.0 PL=0
MOVL C00285 V=800.0 PL=0
MOVL C00286 V=800.0 PL=0
MOVL C00287 V=800.0 PL=0
MOVL C00288 V=800.0 PL=0
MOVL C00289 V=800.0 PL=0
MOVL C00290 V=800.0 PL=0
MOVL C00291 V=800.0 PL=0
MOVL C00292 V=800.0 PL=0
MOVL C00293 V=800.0 PL=0
MOVL C00294 V=800.0 PL=0
MOVL C00295 V=800.0 PL=0
MOVL C00296 V=800.0 PL=0
MOVL C00297 V=800.0 PL=0
MOVL C00298 V=800.0 PL=0
MOVL C00299 V=800.0 PL=0
MOVL C00300 V=800.0 PL=0
MOVL C00301 V=800.0 PL=0
MOVL C00302 V=800.0 PL=0
MOVL C00303 V=800.0 PL=0
MOVL C00304 V=800.0 PL=0
MOVL C00305 V=800.0 PL=0
MOVL C00306 V=800.0 PL=0
MOVL C00307 V=800.0 PL=0
MOVL C00308 V=800.0 PL=0
MOVL C00309 V=800.0 PL=0
MOVL C00310 V=800.0 PL=0
MOVL C00311 V=800.0 PL=0
MOVL C00312 V=800.0 PL=0
MOVL C00313 V=800.0 PL=0
MOVL C00314 V=800.0 PL=0
MOVL C00315 V=800.0 PL=0
MOVL C00316 V=800.0 PL=0
MOVL C00317 V=800.0 PL=0
MOVL C00318 V=800.0 PL=0
MOVL C00319 V=800.0 PL=0
MOVL C00320 V=800.0 PL=0
MOVL C00321 V=800.0 PL=0
MOVL C00322 V=800.0 PL=0
MOVL C00323 V=800.0 PL=0
MOVL C00324 V=800.0 PL=0
MOVL C00325 V=800.0 PL=0
MOVL C00326 V=800.0 PL=0
MOVL C00327 V=800.0 PL=0
MOVL C00328 V=800.0 PL=0
MOVL C00329 V=800.0 PL=0
MOVL C00330 V=800.0 PL=0
MOVL C00331 V=800.0 PL=0
MOVL C00332 V=800.0 PL=0
MOVL C00333 V=800.0 PL=0
MOVL C00334 V=800.0 PL=0
MOVL C00335 V=800.0 PL=0
MOVL C00336 V=800.0 PL=0
MOVL C00337 V=800.0 PL=0
MOVL C00338 V=800.0 PL=0
MOVL C00339 V=800.0 PL=0
MOVL C00340 V=800.0 PL=0
MOVL C00341 V=800.0 PL=0
MOVL C00342 V=800.0 PL=0
MOVL C00343 V=800.0 PL=0
MOVL C00344 V=800.0 PL=0
MOVL C00345 V=800.0 PL=0
MOVL C00346 V=800.0 PL=0
MOVL C00347 V=800.0 PL=0
MOVL C00348 V=800.0 PL=0
MOVL C00349 V=800.0 PL=0
MOVL C00350 V=800.0 PL=0
MOVL C00351 V=800.0 PL=0
MOVL C00352 V=800.0 PL=0
MOVL C00353 V=800.0 PL=0
MOVL C00354 V=800.0 PL=0
MOVL C00355 V=800.0 PL=0
MOVL C00356 V=800.0 PL=0
MOVL C00357 V=800.0 PL=0
MOVL C00358 V=800.0 PL=0
MOVL C00359 V=800.0 PL=0
MOVL C00360 V=800.0 PL=0
MOVL C00361 V=800.0 PL=0
MOVL C00362 V=800.0 PL=0
MOVL C00363 V=800.0 PL=0
MOVL C00364 V=800.0 PL=0
MOVL C00365 V=800.0 PL=0
MOVL C00366 V=800.0 PL=0
MOVL C00367 V=800.0 PL=0
MOVL C00368 V=800.0 PL=0
MOVL C00369 V=800.0 PL=0
MOVL C00370 V=800.0 PL=0
MOVL C00371 V=800.0 PL=0
MOVL C00372 V=800.0 PL=0
MOVL C00373 V=800.0 PL=0
MOVL C00374 V=800.0 PL=0
MOVL C00375 V=800.0 PL=0
MOVL C00376 V=800.0 PL=0
MOVL C00377 V=800.0 PL=0
MOVL C00378 V=800.0 PL=0
MOVL C00379 V=800.0 PL=0
MOVL C00380 V=800.0 PL=0
MOVL C00381 V=800.0 PL=0
MOVL C00382 V=800.0 PL=0
MOVL C00383 V=800.0 PL=0
MOVL C00384 V=800.0 PL=0
MOVL C00385 V=800.0 PL=0
MOVL C00386 V=800.0 PL=0
MOVL C00387 V=800.0 PL=0
MOVL C00388 V=800.0 PL=0
MOVL C00389 V=800.0 PL=0
MOVL C00390 V=800.0 PL=0
MOVL C00391 V=800.0 PL=0
MOVL C00392 V=800.0 PL=0
MOVL C00393 V=800.0 PL=0
MOVL C00394 V=800.0 PL=0
MOVL C00395 V=800.0 PL=0
MOVL C00396 V=800.0 PL=0
MOVL C00397 V=800.0 PL=0
MOVL C00398 V=800.0 PL=0
MOVL C00399 V=800.0 PL=0
MOVL C00400 V=800.0 PL=0
MOVL C00401 V=800.0 PL=0
MOVL C00402 V=800.0 PL=0
MOVL C00403 V=800.0 PL=0
MOVL C00404 V=800.0 PL=0
MOVL C00405 V=800.0 PL=0
MOVL C00406 V=800.0 PL=0
MOVL C00407 V=800.0 PL=0
MOVL C00408 V=800.0 PL=0
MOVL C00409 V=800.0 PL=0
MOVL C00410 V=800.0 PL=0
MOVL C00411 V=800.0 PL=0
MOVL C00412 V=800.0 PL=0
MOVL C00413 V=800.0 PL=0
MOVL C00414 V=800.0 PL=0
MOVL C00415 V=800.0 PL=0
MOVL C00416 V=800.0 PL=0
MOVL C00417 V=800.0 PL=0
MOVL C00418 V=800.0 PL=0
MOVL C00419 V=800.0 PL=0
MOVL C00420 V=800.0 PL=0
MOVL C00421 V=800.0 PL=0
MOVL C00422 V=800.0 PL=0
MOVL C00423 V=800.0 PL=0
MOVL C00424 V=800.0 PL=0
MOVL C00425 V=800.0 PL=0
MOVL C00426 V=800.0 PL=0
MOVL C00427 V=800.0 PL=0
MOVL C00428 V=800.0 PL=0
MOVL C00429 V=800.0 PL=0
MOVL C00430 V=800.0 PL=0
MOVL C00431 V=800.0 PL=0
MOVL C00432 V=800.0 PL=0
MOVL C00433 V=800.0 PL=0
MOVL C00434 V=800.0 PL=0
MOVL C00435 V=800.0 PL=0
MOVL C00436 V=800.0 PL=0
MOVL C00437 V=800.0 PL=0
MOVL C00438 V=800.0 PL=0
MOVL C00439 V=800.0 PL=0
MOVL C00440 V=800.0 PL=0
MOVL C00441 V=800.0 PL=0
MOVL C00442 V=800.0 PL=0
MOVL C00443 V=800.0 PL=0
MOVL C00444 V=800.0 PL=0
MOVL C00445 V=800.0 PL=0
MOVL C00446 V=800.0 PL=0
MOVL C00447 V=800.0 PL=0
MOVL C00448 V=800.0 PL=0
MOVL C00449 V=800.0 PL=0
MOVL C00450 V=800.0 PL=0
MOVL C00451 V=800.0 PL=0
MOVL C00452 V=800.0 PL=0
MOVL C00453 V=800.0 PL=0
MOVL C00454 V=800.0 PL=0
MOVL C00455 V=800.0 PL=0
MOVL C00456 V=800.0 PL=0
MOVL C00457 V=800.0 PL=0
MOVL C00458 V=800.0 PL=0
MOVL C00459 V=800.0 PL=0
MOVL C00460 V=800.0 PL=0
MOVL C00461 V=800.0 PL=0
MOVL C00462 V=800.0 PL=0
MOVL C00463 V=800.0 PL=0
MOVL C00464 V=800.0 PL=0
MOVL C00465 V=800.0 PL=0
MOVL C00466 V=800.0 PL=0
MOVL C00467 V=800.0 PL=0
MOVL C00468 V=800.0 PL=0
MOVL C00469 V=800.0 PL=0
MOVL C00470 V=800.0 PL=0
MOVL C00471 V=800.0 PL=0
MOVL C00472 V=800.0 PL=0
MOVL C00473 V=800.0 PL=0
MOVL C00474 V=800.0 PL=0
MOVL C00475 V=800.0 PL=0
MOVL C00476 V=800.0 PL=0
MOVL C00477 V=800.0 PL=0
MOVL C00478 V=800.0 PL=0
MOVL C00479 V=800.0 PL=0
MOVL C00480 V=800.0 PL=0
MOVL C00481 V=800.0 PL=0
MOVL C00482 V=800.0 PL=0
MOVL C00483 V=800.0 PL=0
MOVL C00484 V=800.0 PL=0
MOVL C00485 V=800.0 PL=0
MOVL C00486 V=800.0 PL=0
MOVL C00487 V=800.0 PL=0
MOVL C00488 V=800.0 PL=0
MOVL C00489 V=800.0 PL=0
MOVL C00490 V=800.0 PL=0
MOVL C00491 V=800.0 PL=0
MOVL C00492 V=800.0 PL=0
MOVL C00493 V=800.0 PL=0
MOVL C00494 V=800.0 PL=0
MOVL C00495 V=800.0 PL=0
MOVL C00496 V=800.0 PL=0
MOVL C00497 V=800.0 PL=0
MOVL C00498 V=800.0 PL=0
MOVL C00499 V=800.0 PL=0
MOVL C00500 V=800.0 PL=0
MOVL C00501 V=800.0 PL=0
MOVL C00502 V=800.0 PL=0
MOVL C00503 V=800.0 PL=0
MOVL C00504 V=800.0 PL=0
MOVL C00505 V=800.0 PL=0
MOVL C00506 V=800.0 PL=0
MOVL C00507 V=800.0 PL=0
MOVL C00508 V=800.0 PL=0
MOVL C00509 V=800.0 PL=0
MOVL C00510 V=800.0 PL=0
MOVL C00511 V=800.0 PL=0
MOVL C00512 V=800.0 PL=0
MOVL C00513 V=800.0 PL=0
MOVL C00514 V=800.0 PL=0
MOVL C00515 V=800.0 PL=0
MOVL C00516 V=800.0 PL=0
MOVL C00517 V=800.0 PL=0
MOVL C00518 V=800.0 PL=0
MOVL C00519 V=800.0 PL=0
MOVL C00520 V=800.0 PL=0
MOVL C00521 V=800.0 PL=0
MOVL C00522 V=800.0 PL=0
MOVL C00523 V=800.0 PL=0
MOVL C00524 V=800.0 PL=0
MOVL C00525 V=800.0 PL=0
MOVL C00526 V=800.0 PL=0
MOVL C00527 V=800.0 PL=0
MOVL C00528 V=800.0 PL=0
MOVL C00529 V=800.0 PL=0
MOVL C00530 V=800.0 PL=0
MOVL C00531 V=800.0 PL=0
MOVL C00532 V=800.0 PL=0
MOVL C00533 V=800.0 PL=0
MOVL C00534 V=800.0 PL=0
MOVL C00535 V=800.0 PL=0
MOVL C00536 V=800.0 PL=0
MOVL C00537 V=800.0 PL=0
MOVL C00538 V=800.0 PL=0
MOVL C00539 V=800.0 PL=0
MOVL C00540 V=800.0 PL=0
MOVL C00541 V=800.0 PL=0
MOVL C00542 V=800.0 PL=0
MOVL C00543 V=800.0 PL=0
MOVL C00544 V=800.0 PL=0
MOVL C00545 V=800.0 PL=0
MOVL C00546 V=800.0 PL=0
MOVL C00547 V=800.0 PL=0
MOVL C00548 V=800.0 PL=0
MOVL C00549 V=800.0 PL=0
MOVL C00550 V=800.0 PL=0
MOVL C00551 V=800.0 PL=0
MOVL C00552 V=800.0 PL=0
MOVL C00553 V=800.0 PL=0
MOVL C00554 V=800.0 PL=0
MOVL C00555 V=800.0 PL=0
MOVL C00556 V=800.0 PL=0
MOVL C00557 V=800.0 PL=0
MOVL C00558 V=800.0 PL=0
MOVL C00559 V=800.0 PL=0
MOVL C00560 V=800.0 PL=0
MOVL C00561 V=800.0 PL=0
MOVL C00562 V=800.0 PL=0
MOVL C00563 V=800.0 PL=0
MOVL C00564 V=800.0 PL=0
MOVL C00565 V=800.0 PL=0
MOVL C00566 V=800.0 PL=0
MOVL C00567 V=800.0 PL=0
MOVL C00568 V=800.0 PL=0
MOVL C00569 V=800.0 PL=0
MOVL C00570 V=800.0 PL=0
MOVL C00571 V=800.0 PL=0
MOVL C00572 V=800.0 PL=0
MOVL C00573 V=800.0 PL=0
MOVL C00574 V=800.0 PL=0
MOVL C00575 V=800.0 PL=0
MOVL C00576 V=800.0 PL=0
MOVL C00577 V=800.0 PL=0
MOVL C00578 V=800.0 PL=0
MOVL C00579 V=800.0 PL=0
MOVL C00580 V=800.0 PL=0
MOVL C00581 V=800.0 PL=0
MOVL C00582 V=800.0 PL=0
MOVL C00583 V=800.0 PL=0
MOVL C00584 V=800.0 PL=0
MOVL C00585 V=800.0 PL=0
MOVL C00586 V=800.0 PL=0
MOVL C00587 V=800.0 PL=0
MOVL C00588 V=800.0 PL=0
MOVL C00589 V=800.0 PL=0
MOVL C00590 V=800.0 PL=0
MOVL C00591 V=800.0 PL=0
MOVL C00592 V=800.0 PL=0
MOVL C00593 V=800.0 PL=0
MOVL C00594 V=800.0 PL=0
MOVL C00595 V=800.0 PL=0
MOVL C00596 V=800.0 PL=0
MOVL C00597 V=800.0 PL=0
MOVL C00598 V=800.0 PL=0
MOVL C00599 V=800.0 PL=0
MOVL C00600 V=800.0 PL=0
MOVL C00601 V=800.0 PL=0
MOVL C00602 V=800.0 PL=0
MOVL C00603 V=800.0 PL=0
MOVL C00604 V=800.0 PL=0
MOVL C00605 V=800.0 PL=0
MOVL C00606 V=800.0 PL=0
MOVL C00607 V=800.0 PL=0
MOVL C00608 V=800.0 PL=0
MOVL C00609 V=800.0 PL=0
MOVL C00610 V=800.0 PL=0
MOVL C00611 V=800.0 PL=0
MOVL C00612 V=800.0 PL=0
MOVL C00613 V=800.0 PL=0
MOVL C00614 V=800.0 PL=0
MOVL C00615 V=800.0 PL=0
MOVL C00616 V=800.0 PL=0
MOVL C00617 V=800.0 PL=0
MOVL C00618 V=800.0 PL=0
MOVL C00619 V=800.0 PL=0
MOVL C00620 V=800.0 PL=0
MOVL C00621 V=800.0 PL=0
MOVL C00622 V=800.0 PL=0
MOVL C00623 V=800.0 PL=0
MOVL C00624 V=800.0 PL=0
MOVL C00625 V=800.0 PL=0
MOVL C00626 V=800.0 PL=0
MOVL C00627 V=800.0 PL=0
MOVL C00628 V=800.0 PL=0
MOVL C00629 V=800.0 PL=0
MOVL C00630 V=800.0 PL=0
MOVL C00631 V=800.0 PL=0
MOVL C00632 V=800.0 PL=0
MOVL C00633 V=800.0 PL=0
MOVL C00634 V=800.0 PL=0
MOVL C00635 V=800.0 PL=0
MOVL C00636 V=800.0 PL=0
MOVL C00637 V=800.0 PL=0
MOVL C00638 V=800.0 PL=0
MOVL C00639 V=800.0 PL=0
MOVL C00640 V=800.0 PL=0
MOVL C00641 V=800.0 PL=0
MOVL C00642 V=800.0 PL=0
MOVL C00643 V=800.0 PL=0
MOVL C00644 V=800.0 PL=0
MOVL C00645 V=800.0 PL=0
MOVL C00646 V=800.0 PL=0
MOVL C00647 V=800.0 PL=0
MOVL C00648 V=800.0 PL=0
MOVL C00649 V=800.0 PL=0
MOVL C00650 V=800.0 PL=0
MOVL C00651 V=800.0 PL=0
MOVL C00652 V=800.0 PL=0
MOVL C00653 V=800.0 PL=0
MOVL C00654 V=800.0 PL=0
MOVL C00655 V=800.0 PL=0
MOVL C00656 V=800.0 PL=0
MOVL C00657 V=800.0 PL=0
MOVL C00658 V=800.0 PL=0
MOVL C00659 V=800.0 PL=0
MOVL C00660 V=800.0 PL=0
MOVL C00661 V=800.0 PL=0
MOVL C00662 V=800.0 PL=0
MOVL C00663 V=800.0 PL=0
MOVL C00664 V=800.0 PL=0
MOVL C00665 V=800.0 PL=0
MOVL C00666 V=800.0 PL=0
MOVL C00667 V=800.0 PL=0
MOVL C00668 V=800.0 PL=0
MOVL C00669 V=800.0 PL=0
MOVL C00670 V=800.0 PL=0
MOVL C00671 V=800.0 PL=0
MOVL C00672 V=800.0 PL=0
MOVL C00673 V=800.0 PL=0
MOVL C00674 V=800.0 PL=0
MOVL C00675 V=800.0 PL=0
MOVL C00676 V=800.0 PL=0
MOVL C00677 V=800.0 PL=0
MOVL C00678 V=800.0 PL=0
MOVL C00679 V=800.0 PL=0
MOVL C00680 V=800.0 PL=0
MOVL C00681 V=800.0 PL=0
MOVL C00682 V=800.0 PL=0
MOVL C00683 V=800.0 PL=0
MOVL C00684 V=800.0 PL=0
MOVL C00685 V=800.0 PL=0
MOVL C00686 V=800.0 PL=0
MOVL C00687 V=800.0 PL=0
MOVL C00688 V=800.0 PL=0
MOVL C00689 V=800.0 PL=0
MOVL C00690 V=800.0 PL=0
MOVL C00691 V=800.0 PL=0
MOVL C00692 V=800.0 PL=0
MOVL C00693 V=800.0 PL=0
MOVL C00694 V=800.0 PL=0
MOVL C00695 V=800.0 PL=0
MOVL C00696 V=800.0 PL=0
MOVL C00697 V=800.0 PL=0
MOVL C00698 V=800.0 PL=0
MOVL C00699 V=800.0 PL=0
MOVL C00700 V=800.0 PL=0
MOVL C00701 V=800.0 PL=0
MOVL C00702 V=800.0 PL=0
MOVL C00703 V=800.0 PL=0
MOVL C00704 V=800.0 PL=0
MOVL C00705 V=800.0 PL=0
MOVL C00706 V=800.0 PL=0
MOVL C00707 V=800.0 PL=0
MOVL C00708 V=800.0 PL=0
MOVL C00709 V=800.0 PL=0
MOVL C00710 V=800.0 PL=0
MOVL C00711 V=800.0 PL=0
MOVL C00712 V=800.0 PL=0
MOVL C00713 V=800.0 PL=0
MOVL C00714 V=800.0 PL=0
MOVL C00715 V=800.0 PL=0
MOVL C00716 V=800.0 PL=0
MOVL C00717 V=800.0 PL=0
MOVL C00718 V=800.0 PL=0
MOVL C00719 V=800.0 PL=0
MOVL C00720 V=800.0 PL=0
MOVL C00721 V=800.0 PL=0
MOVL C00722 V=800.0 PL=0
MOVL C00723 V=800.0 PL=0
MOVL C00724 V=800.0 PL=0
MOVL C00725 V=800.0 PL=0
MOVL C00726 V=800.0 PL=0
MOVL C00727 V=800.0 PL=0
MOVL C00728 V=800.0 PL=0
MOVL C00729 V=800.0 PL=0
MOVL C00730 V=800.0 PL=0
MOVL C00731 V=800.0 PL=0
MOVL C00732 V=800.0 PL=0
MOVL C00733 V=800.0 PL=0
MOVL C00734 V=800.0 PL=0
MOVL C00735 V=800.0 PL=0
MOVL C00736 V=800.0 PL=0
MOVL C00737 V=800.0 PL=0
MOVL C00738 V=800.0 PL=0
MOVL C00739 V=800.0 PL=0
MOVL C00740 V=800.0 PL=0
MOVL C00741 V=800.0 PL=0
MOVL C00742 V=800.0 PL=0
MOVL C00743 V=800.0 PL=0
MOVL C00744 V=800.0 PL=0
MOVL C00745 V=800.0 PL=0
MOVL C00746 V=800.0 PL=0
MOVL C00747 V=800.0 PL=0
MOVL C00748 V=800.0 PL=0
MOVL C00749 V=800.0 PL=0
MOVL C00750 V=800.0 PL=0
MOVL C00751 V=800.0 PL=0
MOVL C00752 V=800.0 PL=0
MOVL C00753 V=800.0 PL=0
MOVL C00754 V=800.0 PL=0
MOVL C00755 V=800.0 PL=0
MOVL C00756 V=800.0 PL=0
MOVL C00757 V=800.0 PL=0
MOVL C00758 V=800.0 PL=0
MOVL C00759 V=800.0 PL=0
MOVL C00760 V=800.0 PL=0
MOVL C00761 V=800.0 PL=0
MOVL C00762 V=800.0 PL=0
MOVL C00763 V=800.0 PL=0
MOVL C00764 V=800.0 PL=0
MOVL C00765 V=800.0 PL=0
MOVL C00766 V=800.0 PL=0
MOVL C00767 V=800.0 PL=0
MOVL C00768 V=800.0 PL=0
MOVL C00769 V=800.0 PL=0
MOVL C00770 V=800.0 PL=0
MOVL C00771 V=800.0 PL=0
MOVL C00772 V=800.0 PL=0
MOVL C00773 V=800.0 PL=0
MOVL C00774 V=800.0 PL=0
MOVL C00775 V=800.0 PL=0
MOVL C00776 V=800.0 PL=0
MOVL C00777 V=800.0 PL=0
MOVL C00778 V=800.0 PL=0
MOVL C00779 V=800.0 PL=0
MOVL C00780 V=800.0 PL=0
MOVL C00781 V=800.0 PL=0
MOVL C00782 V=800.0 PL=0
MOVL C00783 V=800.0 PL=0
MOVL C00784 V=800.0 PL=0
MOVL C00785 V=800.0 PL=0
MOVL C00786 V=800.0 PL=0
MOVL C00787 V=800.0 PL=0
MOVL C00788 V=800.0 PL=0
MOVL C00789 V=800.0 PL=0
MOVL C00790 V=800.0 PL=0
MOVL C00791 V=800.0 PL=0
MOVL C00792 V=800.0 PL=0
MOVL C00793 V=800.0 PL=0
MOVL C00794 V=800.0 PL=0
MOVL C00795 V=800.0 PL=0
MOVL C00796 V=800.0 PL=0
MOVL C00797 V=800.0 PL=0
MOVL C00798 V=800.0 PL=0
MOVL C00799 V=800.0 PL=0
MOVL C00800 V=800.0 PL=0
MOVL C00801 V=800.0 PL=0
MOVL C00802 V=800.0 PL=0
MOVL C00803 V=800.0 PL=0
MOVL C00804 V=800.0 PL=0
MOVL C00805 V=800.0 PL=0
MOVL C00806 V=800.0 PL=0
MOVL C00807 V=800.0 PL=0
MOVL C00808 V=800.0 PL=0
MOVL C00809 V=800.0 PL=0
MOVL C00810 V=800.0 PL=0
MOVL C00811 V=800.0 PL=0
MOVL C00812 V=800.0 PL=0
MOVL C00813 V=800.0 PL=0
MOVL C00814 V=800.0 PL=0
MOVL C00815 V=800.0 PL=0
MOVL C00816 V=800.0 PL=0
MOVL C00817 V=800.0 PL=0
MOVL C00818 V=800.0 PL=0
MOVL C00819 V=800.0 PL=0
MOVL C00820 V=800.0 PL=0
MOVL C00821 V=800.0 PL=0
MOVL C00822 V=800.0 PL=0
MOVL C00823 V=800.0 PL=0
MOVL C00824 V=800.0 PL=0
MOVL C00825 V=800.0 PL=0
MOVL C00826 V=800.0 PL=0
MOVL C00827 V=800.0 PL=0
MOVL C00828 V=800.0 PL=0
MOVL C00829 V=800.0 PL=0
MOVL C00830 V=800.0 PL=0
MOVL C00831 V=800.0 PL=0
MOVL C00832 V=800.0 PL=0
MOVL C00833 V=800.0 PL=0
MOVL C00834 V=800.0 PL=0
MOVL C00835 V=800.0 PL=0
MOVL C00836 V=800.0 PL=0
MOVL C00837 V=800.0 PL=0
MOVL C00838 V=800.0 PL=0
MOVL C00839 V=800.0 PL=0
MOVL C00840 V=800.0 PL=0
MOVL C00841 V=800.0 PL=0
MOVL C00842 V=800.0 PL=0
MOVL C00843 V=800.0 PL=0
MOVL C00844 V=800.0 PL=0
MOVL C00845 V=800.0 PL=0
MOVL C00846 V=800.0 PL=0
MOVL C00847 V=800.0 PL=0
MOVL C00848 V=800.0 PL=0
MOVL C00849 V=800.0 PL=0
MOVL C00850 V=800.0 PL=0
MOVL C00851 V=800.0 PL=0
MOVL C00852 V=800.0 PL=0
MOVL C00853 V=800.0 PL=0
MOVL C00854 V=800.0 PL=0
MOVL C00855 V=800.0 PL=0
MOVL C00856 V=800.0 PL=0
MOVL C00857 V=800.0 PL=0
MOVL C00858 V=800.0 PL=0
MOVL C00859 V=800.0 PL=0
MOVL C00860 V=800.0 PL=0
MOVL C00861 V=800.0 PL=0
MOVL C00862 V=800.0 PL=0
MOVL C00863 V=800.0 PL=0
MOVL C00864 V=800.0 PL=0
MOVL C00865 V=800.0 PL=0
MOVL C00866 V=800.0 PL=0
MOVL C00867 V=800.0 PL=0
MOVL C00868 V=800.0 PL=0
MOVL C00869 V=800.0 PL=0
MOVL C00870 V=800.0 PL=0
MOVL C00871 V=800.0 PL=0
MOVL C00872 V=800.0 PL=0
MOVL C00873 V=800.0 PL=0
MOVL C00874 V=800.0 PL=0
MOVL C00875 V=800.0 PL=0
MOVL C00876 V=800.0 PL=0
MOVL C00877 V=800.0 PL=0
MOVL C00878 V=800.0 PL=0
MOVL C00879 V=800.0 PL=0
MOVL C00880 V=800.0 PL=0
MOVL C00881 V=800.0 PL=0
MOVL C00882 V=800.0 PL=0
MOVL C00883 V=800.0 PL=0
MOVL C00884 V=800.0 PL=0
MOVL C00885 V=800.0 PL=0
MOVL C00886 V=800.0 PL=0
MOVL C00887 V=800.0 PL=0
MOVL C00888 V=800.0 PL=0
MOVL C00889 V=800.0 PL=0
MOVL C00890 V=800.0 PL=0
MOVL C00891 V=800.0 PL=0
MOVL C00892 V=800.0 PL=0
MOVL C00893 V=800.0 PL=0
MOVL C00894 V=800.0 PL=0
MOVL C00895 V=800.0 PL=0
MOVL C00896 V=800.0 PL=0
MOVL C00897 V=800.0 PL=0
MOVL C00898 V=800.0 PL=0
MOVL C00899 V=800.0 PL=0
MOVL C00900 V=800.0 PL=0
MOVL C00901 V=800.0 PL=0
MOVL C00902 V=800.0 PL=0
MOVL C00903 V=800.0 PL=0
MOVL C00904 V=800.0 PL=0
MOVL C00905 V=800.0 PL=0
MOVL C00906 V=800.0 PL=0
MOVL C00907 V=800.0 PL=0
MOVL C00908 V=800.0 PL=0
MOVL C00909 V=800.0 PL=0
MOVL C00910 V=800.0 PL=0
MOVL C00911 V=800.0 PL=0
MOVL C00912 V=800.0 PL=0
MOVL C00913 V=800.0 PL=0
MOVL C00914 V=800.0 PL=0
MOVL C00915 V=800.0 PL=0
MOVL C00916 V=800.0 PL=0
MOVL C00917 V=800.0 PL=0
MOVL C00918 V=800.0 PL=0
MOVL C00919 V=800.0 PL=0
MOVL C00920 V=800.0 PL=0
MOVL C00921 V=800.0 PL=0
MOVL C00922 V=800.0 PL=0
MOVL C00923 V=800.0 PL=0
MOVL C00924 V=800.0 PL=0
MOVL C00925 V=800.0 PL=0
MOVL C00926 V=800.0 PL=0
MOVL C00927 V=800.0 PL=0
MOVL C00928 V=800.0 PL=0
MOVL C00929 V=800.0 PL=0
MOVL C00930 V=800.0 PL=0
MOVL C00931 V=800.0 PL=0
MOVL C00932 V=800.0 PL=0
MOVL C00933 V=800.0 PL=0
MOVL C00934 V=800.0 PL=0
MOVL C00935 V=800.0 PL=0
MOVL C00936 V=800.0 PL=0
MOVL C00937 V=800.0 PL=0
MOVL C00938 V=800.0 PL=0
MOVL C00939 V=800.0 PL=0
MOVL C00940 V=800.0 PL=0
MOVL C00941 V=800.0 PL=0
MOVL C00942 V=800.0 PL=0
MOVL C00943 V=800.0 PL=0
MOVL C00944 V=800.0 PL=0
MOVL C00945 V=800.0 PL=0
MOVL C00946 V=800.0 PL=0
MOVL C00947 V=800.0 PL=0
MOVL C00948 V=800.0 PL=0
MOVL C00949 V=800.0 PL=0
MOVL C00950 V=800.0 PL=0
MOVL C00951 V=800.0 PL=0
MOVL C00952 V=800.0 PL=0
MOVL C00953 V=800.0 PL=0
MOVL C00954 V=800.0 PL=0
MOVL C00955 V=800.0 PL=0
MOVL C00956 V=800.0 PL=0
MOVL C00957 V=800.0 PL=0
MOVL C00958 V=800.0 PL=0
MOVL C00959 V=800.0 PL=0
MOVL C00960 V=800.0 PL=0
MOVL C00961 V=800.0 PL=0
MOVL C00962 V=800.0 PL=0
MOVL C00963 V=800.0 PL=0
MOVL C00964 V=800.0 PL=0
MOVL C00965 V=800.0 PL=0
MOVL C00966 V=800.0 PL=0
MOVL C00967 V=800.0 PL=0
MOVL C00968 V=800.0 PL=0
MOVL C00969 V=800.0 PL=0
MOVL C00970 V=800.0 PL=0
MOVL C00971 V=800.0 PL=0
MOVL C00972 V=800.0 PL=0
MOVL C00973 V=800.0 PL=0
MOVL C00974 V=800.0 PL=0
MOVL C00975 V=800.0 PL=0
MOVL C00976 V=800.0 PL=0
MOVL C00977 V=800.0 PL=0
MOVL C00978 V=800.0 PL=0
MOVL C00979 V=800.0 PL=0
MOVL C00980 V=800.0 PL=0
MOVL C00981 V=800.0 PL=0
MOVL C00982 V=800.0 PL=0
MOVL C00983 V=800.0 PL=0
MOVL C00984 V=800.0 PL=0
MOVL C00985 V=800.0 PL=0
MOVL C00986 V=800.0 PL=0
MOVL C00987 V=800.0 PL=0
MOVL C00988 V=800.0 PL=0
MOVL C00989 V=800.0 PL=0
MOVL C00990 V=800.0 PL=0
MOVL C00991 V=800.0 PL=0
MOVL C00992 V=800.0 PL=0
MOVL C00993 V=800.0 PL=0
MOVL C00994 V=800.0 PL=0
MOVL C00995 V=800.0 PL=0
MOVL C00996 V=800.0 PL=0
MOVL C00997 V=800.0 PL=0
MOVL C00998 V=800.0 PL=0
MOVL C00999 V=800.0 PL=0
MOVL C01000 V=800.0 PL=0
MOVL C01001 V=800.0 PL=0
MOVL C01002 V=800.0 PL=0
MOVL C01003 V=800.0 PL=0
MOVL C01004 V=800.0 PL=0
MOVL C01005 V=800.0 PL=0
MOVL C01006 V=800.0 PL=0
MOVL C01007 V=800.0 PL=0
MOVL C01008 V=800.0 PL=0
MOVL C01009 V=800.0 PL=0
MOVL C01010 V=800.0 PL=0
MOVL C01011 V=800.0 PL=0
MOVL C01012 V=800.0 PL=0
MOVL C01013 V=800.0 PL=0
MOVL C01014 V=800.0 PL=0
MOVL C01015 V=800.0 PL=0
MOVL C01016 V=800.0 PL=0
MOVL C01017 V=800.0 PL=0
MOVL C01018 V=800.0 PL=0
MOVL C01019 V=800.0 PL=0
MOVL C01020 V=800.0 PL=0
MOVL C01021 V=800.0 PL=0
MOVL C01022 V=800.0 PL=0
MOVL C01023 V=800.0 PL=0
MOVL C01024 V=800.0 PL=0
MOVL C01025 V=800.0 PL=0
MOVL C01026 V=800.0 PL=0
MOVL C01027 V=800.0 PL=0
MOVL C01028 V=800.0 PL=0
MOVL C01029 V=800.0 PL=0
MOVL C01030 V=800.0 PL=0
MOVL C01031 V=800.0 PL=0
MOVL C01032 V=800.0 PL=0
MOVL C01033 V=800.0 PL=0
MOVL C01034 V=800.0 PL=0
MOVL C01035 V=800.0 PL=0
MOVL C01036 V=800.0 PL=0
MOVL C01037 V=800.0 PL=0
MOVL C01038 V=800.0 PL=0
MOVL C01039 V=800.0 PL=0
MOVL C01040 V=800.0 PL=0
MOVL C01041 V=800.0 PL=0
MOVL C01042 V=800.0 PL=0
MOVL C01043 V=800.0 PL=0
MOVL C01044 V=800.0 PL=0
MOVL C01045 V=800.0 PL=0
MOVL C01046 V=800.0 PL=0
MOVL C01047 V=800.0 PL=0
MOVL C01048 V=800.0 PL=0
MOVL C01049 V=800.0 PL=0
MOVL C01050 V=800.0 PL=0
MOVL C01051 V=800.0 PL=0
MOVL C01052 V=800.0 PL=0
MOVL C01053 V=800.0 PL=0
MOVL C01054 V=800.0 PL=0
MOVL C01055 V=800.0 PL=0
MOVL C01056 V=800.0 PL=0
MOVL C01057 V=800.0 PL=0
MOVL C01058 V=800.0 PL=0
MOVL C01059 V=800.0 PL=0
MOVL C01060 V=800.0 PL=0
MOVL C01061 V=800.0 PL=0
MOVL C01062 V=800.0 PL=0
MOVL C01063 V=800.0 PL=0
MOVL C01064 V=800.0 PL=0
MOVL C01065 V=800.0 PL=0
MOVL C01066 V=800.0 PL=0
MOVL C01067 V=800.0 PL=0
MOVL C01068 V=800.0 PL=0
MOVL C01069 V=800.0 PL=0
MOVL C01070 V=800.0 PL=0
MOVL C01071 V=800.0 PL=0
MOVL C01072 V=800.0 PL=0
MOVL C01073 V=800.0 PL=0
MOVL C01074 V=800.0 PL=0
MOVL C01075 V=800.0 PL=0
MOVL C01076 V=800.0 PL=0
MOVL C01077 V=800.0 PL=0
MOVL C01078 V=800.0 PL=0
MOVL C01079 V=800.0 PL=0
MOVL C01080 V=800.0 PL=0
MOVL C01081 V=800.0 PL=0
MOVL C01082 V=800.0 PL=0
MOVL C01083 V=800.0 PL=0
MOVL C01084 V=800.0 PL=0
MOVL C01085 V=800.0 PL=0
MOVL C01086 V=800.0 PL=0
MOVL C01087 V=800.0 PL=0
MOVL C01088 V=800.0 PL=0
MOVL C01089 V=800.0 PL=0
MOVL C01090 V=800.0 PL=0
MOVL C01091 V=800.0 PL=0
MOVL C01092 V=800.0 PL=0
MOVL C01093 V=800.0 PL=0
MOVL C01094 V=800.0 PL=0
MOVL C01095 V=800.0 PL=0
MOVL C01096 V=800.0 PL=0
MOVL C01097 V=800.0 PL=0
MOVL C01098 V=800.0 PL=0
MOVL C01099 V=800.0 PL=0
MOVL C01100 V=800.0 PL=0
MOVL C01101 V=800.0 PL=0
MOVL C01102 V=800.0 PL=0
MOVL C01103 V=800.0 PL=0
MOVL C01104 V=800.0 PL=0
MOVL C01105 V=800.0 PL=0
MOVL C01106 V=800.0 PL=0
MOVL C01107 V=800.0 PL=0
MOVL C01108 V=800.0 PL=0
MOVL C01109 V=800.0 PL=0
MOVL C01110 V=800.0 PL=0
MOVL C01111 V=800.0 PL=0
MOVL C01112 V=800.0 PL=0
MOVL C01113 V=800.0 PL=0
MOVL C01114 V=800.0 PL=0
MOVL C01115 V=800.0 PL=0
MOVL C01116 V=800.0 PL=0
MOVL C01117 V=800.0 PL=0
MOVL C01118 V=800.0 PL=0
MOVL C01119 V=800.0 PL=0
MOVL C01120 V=800.0 PL=0
MOVL C01121 V=800.0 PL=0
MOVL C01122 V=800.0 PL=0
MOVL C01123 V=800.0 PL=0
MOVL C01124 V=800.0 PL=0
MOVL C01125 V=800.0 PL=0
MOVL C01126 V=800.0 PL=0
MOVL C01127 V=800.0 PL=0
MOVL C01128 V=800.0 PL=0
MOVL C01129 V=800.0 PL=0
MOVL C01130 V=800.0 PL=0
MOVL C01131 V=800.0 PL=0
MOVL C01132 V=800.0 PL=0
MOVL C01133 V=800.0 PL=0
MOVL C01134 V=800.0 PL=0
MOVL C01135 V=800.0 PL=0
MOVL C01136 V=800.0 PL=0
MOVL C01137 V=800.0 PL=0
MOVL C01138 V=800.0 PL=0
MOVL C01139 V=800.0 PL=0
MOVL C01140 V=800.0 PL=0
MOVL C01141 V=800.0 PL=0
MOVL C01142 V=800.0 PL=0
MOVL C01143 V=800.0 PL=0
MOVL C01144 V=800.0 PL=0
MOVL C01145 V=800.0 PL=0
MOVL C01146 V=800.0 PL=0
MOVL C01147 V=800.0 PL=0
MOVL C01148 V=800.0 PL=0
MOVL C01149 V=800.0 PL=0
MOVL C01150 V=800.0 PL=0
MOVL C01151 V=800.0 PL=0
MOVL C01152 V=800.0 PL=0
MOVL C01153 V=800.0 PL=0
MOVL C01154 V=800.0 PL=0
MOVL C01155 V=800.0 PL=0
MOVL C01156 V=800.0 PL=0
MOVL C01157 V=800.0 PL=0
MOVL C01158 V=800.0 PL=0
MOVL C01159 V=800.0 PL=0
MOVL C01160 V=800.0 PL=0
MOVL C01161 V=800.0 PL=0
MOVL C01162 V=800.0 PL=0
MOVL C01163 V=800.0 PL=0
MOVL C01164 V=800.0 PL=0
MOVL C01165 V=800.0 PL=0
MOVL C01166 V=800.0 PL=0
MOVL C01167 V=800.0 PL=0
MOVL C01168 V=800.0 PL=0
MOVL C01169 V=800.0 PL=0
MOVL C01170 V=800.0 PL=0
MOVL C01171 V=800.0 PL=0
MOVL C01172 V=800.0 PL=0
MOVL C01173 V=800.0 PL=0
MOVL C01174 V=800.0 PL=0
MOVL C01175 V=800.0 PL=0
MOVL C01176 V=800.0 PL=0
MOVL C01177 V=800.0 PL=0
MOVL C01178 V=800.0 PL=0
MOVL C01179 V=800.0 PL=0
MOVL C01180 V=800.0 PL=0
MOVL C01181 V=800.0 PL=0
MOVL C01182 V=800.0 PL=0
MOVL C01183 V=800.0 PL=0
MOVL C01184 V=800.0 PL=0
MOVL C01185 V=800.0 PL=0
MOVL C01186 V=800.0 PL=0
MOVL C01187 V=800.0 PL=0
MOVL C01188 V=800.0 PL=0
MOVL C01189 V=800.0 PL=0
MOVL C01190 V=800.0 PL=0
MOVL C01191 V=800.0 PL=0
MOVL C01192 V=800.0 PL=0
MOVL C01193 V=800.0 PL=0
MOVL C01194 V=800.0 PL=0
MOVL C01195 V=800.0 PL=0
MOVL C01196 V=800.0 PL=0
MOVL C01197 V=800.0 PL=0
MOVL C01198 V=800.0 PL=0
MOVL C01199 V=800.0 PL=0
MOVL C01200 V=800.0 PL=0
MOVL C01201 V=800.0 PL=0
MOVL C01202 V=800.0 PL=0
MOVL C01203 V=800.0 PL=0
MOVL C01204 V=800.0 PL=0
MOVL C01205 V=800.0 PL=0
MOVL C01206 V=800.0 PL=0
MOVL C01207 V=800.0 PL=0
MOVL C01208 V=800.0 PL=0
MOVL C01209 V=800.0 PL=0
MOVL C01210 V=800.0 PL=0
MOVL C01211 V=800.0 PL=0
MOVL C01212 V=800.0 PL=0
MOVL C01213 V=800.0 PL=0
MOVL C01214 V=800.0 PL=0
MOVL C01215 V=800.0 PL=0
MOVL C01216 V=800.0 PL=0
MOVL C01217 V=800.0 PL=0
MOVL C01218 V=800.0 PL=0
MOVL C01219 V=800.0 PL=0
MOVL C01220 V=800.0 PL=0
MOVL C01221 V=800.0 PL=0
MOVL C01222 V=800.0 PL=0
MOVL C01223 V=800.0 PL=0
MOVL C01224 V=800.0 PL=0
MOVL C01225 V=800.0 PL=0
MOVL C01226 V=800.0 PL=0
MOVL C01227 V=800.0 PL=0
MOVL C01228 V=800.0 PL=0
MOVL C01229 V=800.0 PL=0
MOVL C01230 V=800.0 PL=0
MOVL C01231 V=800.0 PL=0
MOVL C01232 V=800.0 PL=0
MOVL C01233 V=800.0 PL=0
MOVL C01234 V=800.0 PL=0
MOVL C01235 V=800.0 PL=0
MOVL C01236 V=800.0 PL=0
MOVL C01237 V=800.0 PL=0
MOVL C01238 V=800.0 PL=0
MOVL C01239 V=800.0 PL=0
MOVL C01240 V=800.0 PL=0
MOVL C01241 V=800.0 PL=0
MOVL C01242 V=800.0 PL=0
MOVL C01243 V=800.0 PL=0
MOVL C01244 V=800.0 PL=0
MOVL C01245 V=800.0 PL=0
MOVL C01246 V=800.0 PL=0
MOVL C01247 V=800.0 PL=0
MOVL C01248 V=800.0 PL=0
MOVL C01249 V=800.0 PL=0
MOVL C01250 V=800.0 PL=0
MOVL C01251 V=800.0 PL=0
MOVL C01252 V=800.0 PL=0
MOVL C01253 V=800.0 PL=0
MOVL C01254 V=800.0 PL=0
MOVL C01255 V=800.0 PL=0
MOVL C01256 V=800.0 PL=0
MOVL C01257 V=800.0 PL=0
MOVL C01258 V=800.0 PL=0
MOVL C01259 V=800.0 PL=0
MOVL C01260 V=800.0 PL=0
MOVL C01261 V=800.0 PL=0
MOVL C01262 V=800.0 PL=0
MOVL C01263 V=800.0 PL=0
MOVL C01264 V=800.0 PL=0
MOVL C01265 V=800.0 PL=0
MOVL C01266 V=800.0 PL=0
MOVL C01267 V=800.0 PL=0
MOVL C01268 V=800.0 PL=0
MOVL C01269 V=800.0 PL=0
MOVL C01270 V=800.0 PL=0
MOVL C01271 V=800.0 PL=0
MOVL C01272 V=800.0 PL=0
MOVL C01273 V=800.0 PL=0
MOVL C01274 V=800.0 PL=0
MOVL C01275 V=800.0 PL=0
MOVL C01276 V=800.0 PL=0
MOVL C01277 V=800.0 PL=0
MOVL C01278 V=800.0 PL=0
MOVL C01279 V=800.0 PL=0
MOVL C01280 V=800.0 PL=0
MOVL C01281 V=800.0 PL=0
MOVL C01282 V=800.0 PL=0
MOVL C01283 V=800.0 PL=0
MOVL C01284 V=800.0 PL=0
MOVL C01285 V=800.0 PL=0
MOVL C01286 V=800.0 PL=0
MOVL C01287 V=800.0 PL=0
MOVL C01288 V=800.0 PL=0
MOVL C01289 V=800.0 PL=0
MOVL C01290 V=800.0 PL=0
MOVL C01291 V=800.0 PL=0
MOVL C01292 V=800.0 PL=0
MOVL C01293 V=800.0 PL=0
MOVL C01294 V=800.0 PL=0
MOVL C01295 V=800.0 PL=0
MOVL C01296 V=800.0 PL=0
MOVL C01297 V=800.0 PL=0
MOVL C01298 V=800.0 PL=0
MOVL C01299 V=800.0 PL=0
MOVL C01300 V=800.0 PL=0
MOVL C01301 V=800.0 PL=0
MOVL C01302 V=800.0 PL=0
MOVL C01303 V=800.0 PL=0
MOVL C01304 V=800.0 PL=0
MOVL C01305 V=800.0 PL=0
MOVL C01306 V=800.0 PL=0
MOVL C01307 V=800.0 PL=0
MOVL C01308 V=800.0 PL=0
MOVL C01309 V=800.0 PL=0
MOVL C01310 V=800.0 PL=0
MOVL C01311 V=800.0 PL=0
MOVL C01312 V=800.0 PL=0
MOVL C01313 V=800.0 PL=0
MOVL C01314 V=800.0 PL=0
MOVL C01315 V=800.0 PL=0
MOVL C01316 V=800.0 PL=0
MOVL C01317 V=800.0 PL=0
MOVL C01318 V=800.0 PL=0
MOVL C01319 V=800.0 PL=0
MOVL C01320 V=800.0 PL=0
MOVL C01321 V=800.0 PL=0
MOVL C01322 V=800.0 PL=0
MOVL C01323 V=800.0 PL=0
MOVL C01324 V=800.0 PL=0
MOVL C01325 V=800.0 PL=0
MOVL C01326 V=800.0 PL=0
MOVL C01327 V=800.0 PL=0
MOVL C01328 V=800.0 PL=0
MOVL C01329 V=800.0 PL=0
MOVL C01330 V=800.0 PL=0
MOVL C01331 V=800.0 PL=0
MOVL C01332 V=800.0 PL=0
MOVL C01333 V=800.0 PL=0
MOVL C01334 V=800.0 PL=0
MOVL C01335 V=800.0 PL=0
MOVL C01336 V=800.0 PL=0
MOVL C01337 V=800.0 PL=0
MOVL C01338 V=800.0 PL=0
MOVL C01339 V=800.0 PL=0
MOVL C01340 V=800.0 PL=0
MOVL C01341 V=800.0 PL=0
MOVL C01342 V=800.0 PL=0
MOVL C01343 V=800.0 PL=0
MOVL C01344 V=800.0 PL=0
MOVL C01345 V=800.0 PL=0
MOVL C01346 V=800.0 PL=0
MOVL C01347 V=800.0 PL=0
MOVL C01348 V=800.0 PL=0
MOVL C01349 V=800.0 PL=0
MOVL C01350 V=800.0 PL=0
MOVL C01351 V=800.0 PL=0
MOVL C01352 V=800.0 PL=0
MOVL C01353 V=800.0 PL=0
MOVL C01354 V=800.0 PL=0
MOVL C01355 V=800.0 PL=0
MOVL C01356 V=800.0 PL=0
MOVL C01357 V=800.0 PL=0
MOVL C01358 V=800.0 PL=0
MOVL C01359 V=800.0 PL=0
MOVL C01360 V=800.0 PL=0
MOVL C01361 V=800.0 PL=0
MOVL C01362 V=800.0 PL=0
MOVL C01363 V=800.0 PL=0
MOVL C01364 V=800.0 PL=0
MOVL C01365 V=800.0 PL=0
MOVL C01366 V=800.0 PL=0
MOVL C01367 V=800.0 PL=0
MOVL C01368 V=800.0 PL=0
MOVL C01369 V=800.0 PL=0
MOVL C01370 V=800.0 PL=0
MOVL C01371 V=800.0 PL=0
MOVL C01372 V=800.0 PL=0
MOVL C01373 V=800.0 PL=0
MOVL C01374 V=800.0 PL=0
MOVL C01375 V=800.0 PL=0
MOVL C01376 V=800.0 PL=0
MOVL C01377 V=800.0 PL=0
MOVL C01378 V=800.0 PL=0
MOVL C01379 V=800.0 PL=0
MOVL C01380 V=800.0 PL=0
MOVL C01381 V=800.0 PL=0
MOVL C01382 V=800.0 PL=0
MOVL C01383 V=800.0 PL=0
MOVL C01384 V=800.0 PL=0
MOVL C01385 V=800.0 PL=0
MOVL C01386 V=800.0 PL=0
MOVL C01387 V=800.0 PL=0
MOVL C01388 V=800.0 PL=0
MOVL C01389 V=800.0 PL=0
MOVL C01390 V=800.0 PL=0
MOVL C01391 V=800.0 PL=0
MOVL C01392 V=800.0 PL=0
MOVL C01393 V=800.0 PL=0
MOVL C01394 V=800.0 PL=0
MOVL C01395 V=800.0 PL=0
MOVL C01396 V=800.0 PL=0
MOVL C01397 V=800.0 PL=0
MOVL C01398 V=800.0 PL=0
MOVL C01399 V=800.0 PL=0
MOVL C01400 V=800.0 PL=0
MOVL C01401 V=800.0 PL=0
MOVL C01402 V=800.0 PL=0
MOVL C01403 V=800.0 PL=0
MOVL C01404 V=800.0 PL=0
MOVL C01405 V=800.0 PL=0
MOVL C01406 V=800.0 PL=0
MOVL C01407 V=800.0 PL=0
MOVL C01408 V=800.0 PL=0
MOVL C01409 V=800.0 PL=0
MOVL C01410 V=800.0 PL=0
MOVL C01411 V=800.0 PL=0
MOVL C01412 V=800.0 PL=0
MOVL C01413 V=800.0 PL=0
MOVL C01414 V=800.0 PL=0
MOVL C01415 V=800.0 PL=0
MOVL C01416 V=800.0 PL=0
MOVL C01417 V=800.0 PL=0
MOVL C01418 V=800.0 PL=0
MOVL C01419 V=800.0 PL=0
MOVL C01420 V=800.0 PL=0
MOVL C01421 V=800.0 PL=0
MOVL C01422 V=800.0 PL=0
MOVL C01423 V=800.0 PL=0
MOVL C01424 V=800.0 PL=0
MOVL C01425 V=800.0 PL=0
MOVL C01426 V=800.0 PL=0
MOVL C01427 V=800.0 PL=0
MOVL C01428 V=800.0 PL=0
MOVL C01429 V=800.0 PL=0
MOVL C01430 V=800.0 PL=0
MOVL C01431 V=800.0 PL=0
MOVL C01432 V=800.0 PL=0
MOVL C01433 V=800.0 PL=0
MOVL C01434 V=800.0 PL=0
MOVL C01435 V=800.0 PL=0
MOVL C01436 V=800.0 PL=0
MOVL C01437 V=800.0 PL=0
MOVL C01438 V=800.0 PL=0
MOVL C01439 V=800.0 PL=0
MOVL C01440 V=800.0 PL=0
MOVL C01441 V=800.0 PL=0
MOVL C01442 V=800.0 PL=0
MOVL C01443 V=800.0 PL=0
MOVL C01444 V=800.0 PL=0
MOVL C01445 V=800.0 PL=0
MOVL C01446 V=800.0 PL=0
MOVL C01447 V=800.0 PL=0
MOVL C01448 V=800.0 PL=0
MOVL C01449 V=800.0 PL=0
MOVL C01450 V=800.0 PL=0
MOVL C01451 V=800.0 PL=0
MOVL C01452 V=800.0 PL=0
MOVL C01453 V=800.0 PL=0
MOVL C01454 V=800.0 PL=0
MOVL C01455 V=800.0 PL=0
MOVL C01456 V=800.0 PL=0
MOVL C01457 V=800.0 PL=0
MOVL C01458 V=800.0 PL=0
MOVL C01459 V=800.0 PL=0
MOVL C01460 V=800.0 PL=0
MOVL C01461 V=800.0 PL=0
MOVL C01462 V=800.0 PL=0
MOVL C01463 V=800.0 PL=0
MOVL C01464 V=800.0 PL=0
MOVL C01465 V=800.0 PL=0
MOVL C01466 V=800.0 PL=0
MOVL C01467 V=800.0 PL=0
MOVL C01468 V=800.0 PL=0
MOVL C01469 V=800.0 PL=0
MOVL C01470 V=800.0 PL=0
MOVL C01471 V=800.0 PL=0
MOVL C01472 V=800.0 PL=0
MOVL C01473 V=800.0 PL=0
MOVL C01474 V=800.0 PL=0
MOVL C01475 V=800.0 PL=0
MOVL C01476 V=800.0 PL=0
MOVL C01477 V=800.0 PL=0
MOVL C01478 V=800.0 PL=0
MOVL C01479 V=800.0 PL=0
MOVL C01480 V=800.0 PL=0
MOVL C01481 V=800.0 PL=0
MOVL C01482 V=800.0 PL=0
MOVL C01483 V=800.0 PL=0
MOVL C01484 V=800.0 PL=0
MOVL C01485 V=800.0 PL=0
MOVL C01486 V=800.0 PL=0
MOVL C01487 V=800.0 PL=0
MOVL C01488 V=800.0 PL=0
MOVL C01489 V=800.0 PL=0
MOVL C01490 V=800.0 PL=0
MOVL C01491 V=800.0 PL=0
MOVL C01492 V=800.0 PL=0
MOVL C01493 V=800.0 PL=0
MOVL C01494 V=800.0 PL=0
MOVL C01495 V=800.0 PL=0
MOVL C01496 V=800.0 PL=0
MOVL C01497 V=800.0 PL=0
MOVL C01498 V=800.0 PL=0
MOVL C01499 V=800.0 PL=0
MOVL C01500 V=800.0 PL=0
MOVL C01501 V=800.0 PL=0
MOVL C01502 V=800.0 PL=0
MOVL C01503 V=800.0 PL=0
MOVL C01504 V=800.0 PL=0
MOVL C01505 V=800.0 PL=0
MOVL C01506 V=800.0 PL=0
MOVL C01507 V=800.0 PL=0
MOVL C01508 V=800.0 PL=0
MOVL C01509 V=800.0 PL=0
MOVL C01510 V=800.0 PL=0
MOVL C01511 V=800.0 PL=0
MOVL C01512 V=800.0 PL=0
MOVL C01513 V=800.0 PL=0
MOVL C01514 V=800.0 PL=0
MOVL C01515 V=800.0 PL=0
MOVL C01516 V=800.0 PL=0
MOVL C01517 V=800.0 PL=0
MOVL C01518 V=800.0 PL=0
MOVL C01519 V=800.0 PL=0
MOVL C01520 V=800.0 PL=0
MOVL C01521 V=800.0 PL=0
MOVL C01522 V=800.0 PL=0
MOVL C01523 V=800.0 PL=0
MOVL C01524 V=800.0 PL=0
MOVL C01525 V=800.0 PL=0
MOVL C01526 V=800.0 PL=0
MOVL C01527 V=800.0 PL=0
MOVL C01528 V=800.0 PL=0
MOVL C01529 V=800.0 PL=0
MOVL C01530 V=800.0 PL=0
MOVL C01531 V=800.0 PL=0
MOVL C01532 V=800.0 PL=0
MOVL C01533 V=800.0 PL=0
MOVL C01534 V=800.0 PL=0
MOVL C01535 V=800.0 PL=0
MOVL C01536 V=800.0 PL=0
MOVL C01537 V=800.0 PL=0
MOVL C01538 V=800.0 PL=0
MOVL C01539 V=800.0 PL=0
MOVL C01540 V=800.0 PL=0
MOVL C01541 V=800.0 PL=0
MOVL C01542 V=800.0 PL=0
MOVL C01543 V=800.0 PL=0
MOVL C01544 V=800.0 PL=0
MOVL C01545 V=800.0 PL=0
MOVL C01546 V=800.0 PL=0
MOVL C01547 V=800.0 PL=0
MOVL C01548 V=800.0 PL=0
MOVL C01549 V=800.0 PL=0
MOVL C01550 V=800.0 PL=0
MOVL C01551 V=800.0 PL=0
MOVL C01552 V=800.0 PL=0
MOVL C01553 V=800.0 PL=0
MOVL C01554 V=800.0 PL=0
MOVL C01555 V=800.0 PL=0
MOVL C01556 V=800.0 PL=0
MOVL C01557 V=800.0 PL=0
MOVL C01558 V=800.0 PL=0
MOVL C01559 V=800.0 PL=0
MOVL C01560 V=800.0 PL=0
MOVL C01561 V=800.0 PL=0
MOVL C01562 V=800.0 PL=0
MOVL C01563 V=800.0 PL=0
MOVL C01564 V=800.0 PL=0
MOVL C01565 V=800.0 PL=0
MOVL C01566 V=800.0 PL=0
MOVL C01567 V=800.0 PL=0
MOVL C01568 V=800.0 PL=0
MOVL C01569 V=800.0 PL=0
MOVL C01570 V=800.0 PL=0
MOVL C01571 V=800.0 PL=0
MOVL C01572 V=800.0 PL=0
MOVL C01573 V=800.0 PL=0
MOVL C01574 V=800.0 PL=0
MOVL C01575 V=800.0 PL=0
MOVL C01576 V=800.0 PL=0
MOVL C01577 V=800.0 PL=0
MOVL C01578 V=800.0 PL=0
MOVL C01579 V=800.0 PL=0
MOVL C01580 V=800.0 PL=0
MOVL C01581 V=800.0 PL=0
MOVL C01582 V=800.0 PL=0
MOVL C01583 V=800.0 PL=0
MOVL C01584 V=800.0 PL=0
MOVL C01585 V=800.0 PL=0
MOVL C01586 V=800.0 PL=0
MOVL C01587 V=800.0 PL=0
MOVL C01588 V=800.0 PL=0
MOVL C01589 V=800.0 PL=0
MOVL C01590 V=800.0 PL=0
MOVL C01591 V=800.0 PL=0
MOVL C01592 V=800.0 PL=0
MOVL C01593 V=800.0 PL=0
MOVL C01594 V=800.0 PL=0
MOVL C01595 V=800.0 PL=0
MOVL C01596 V=800.0 PL=0
MOVL C01597 V=800.0 PL=0
MOVL C01598 V=800.0 PL=0
MOVL C01599 V=800.0 PL=0
MOVL C01600 V=800.0 PL=0
MOVL C01601 V=800.0 PL=0
MOVL C01602 V=800.0 PL=0
MOVL C01603 V=800.0 PL=0
MOVL C01604 V=800.0 PL=0
MOVL C01605 V=800.0 PL=0
MOVL C01606 V=800.0 PL=0
MOVL C01607 V=800.0 PL=0
MOVL C01608 V=800.0 PL=0
MOVL C01609 V=800.0 PL=0
MOVL C01610 V=800.0 PL=0
MOVL C01611 V=800.0 PL=0
MOVL C01612 V=800.0 PL=0
MOVL C01613 V=800.0 PL=0
MOVL C01614 V=800.0 PL=0
MOVL C01615 V=800.0 PL=0
MOVL C01616 V=800.0 PL=0
MOVL C01617 V=800.0 PL=0
MOVL C01618 V=800.0 PL=0
MOVL C01619 V=800.0 PL=0
MOVL C01620 V=800.0 PL=0
MOVL C01621 V=800.0 PL=0
MOVL C01622 V=800.0 PL=0
MOVL C01623 V=800.0 PL=0
MOVL C01624 V=800.0 PL=0
MOVL C01625 V=800.0 PL=0
MOVL C01626 V=800.0 PL=0
MOVL C01627 V=800.0 PL=0
MOVL C01628 V=800.0 PL=0
MOVL C01629 V=800.0 PL=0
MOVL C01630 V=800.0 PL=0
MOVL C01631 V=800.0 PL=0
MOVL C01632 V=800.0 PL=0
MOVL C01633 V=800.0 PL=0
MOVL C01634 V=800.0 PL=0
MOVL C01635 V=800.0 PL=0
MOVL C01636 V=800.0 PL=0
MOVL C01637 V=800.0 PL=0
MOVL C01638 V=800.0 PL=0
MOVL C01639 V=800.0 PL=0
MOVL C01640 V=800.0 PL=0
MOVL C01641 V=800.0 PL=0
MOVL C01642 V=800.0 PL=0
MOVL C01643 V=800.0 PL=0
MOVL C01644 V=800.0 PL=0
MOVL C01645 V=800.0 PL=0
MOVL C01646 V=800.0 PL=0
MOVL C01647 V=800.0 PL=0
MOVL C01648 V=800.0 PL=0
MOVL C01649 V=800.0 PL=0
MOVL C01650 V=800.0 PL=0
MOVL C01651 V=800.0 PL=0
MOVL C01652 V=800.0 PL=0
MOVL C01653 V=800.0 PL=0
MOVL C01654 V=800.0 PL=0
MOVL C01655 V=800.0 PL=0
MOVL C01656 V=800.0 PL=0
MOVL C01657 V=800.0 PL=0
MOVL C01658 V=800.0 PL=0
MOVL C01659 V=800.0 PL=0
MOVL C01660 V=800.0 PL=0
MOVL C01661 V=800.0 PL=0
MOVL C01662 V=800.0 PL=0
MOVL C01663 V=800.0 PL=0
MOVL C01664 V=800.0 PL=0
MOVL C01665 V=800.0 PL=0
MOVL C01666 V=800.0 PL=0
MOVL C01667 V=800.0 PL=0
MOVL C01668 V=800.0 PL=0
MOVL C01669 V=800.0 PL=0
MOVL C01670 V=800.0 PL=0
MOVL C01671 V=800.0 PL=0
MOVL C01672 V=800.0 PL=0
MOVL C01673 V=800.0 PL=0
MOVL C01674 V=800.0 PL=0
MOVL C01675 V=800.0 PL=0
MOVL C01676 V=800.0 PL=0
MOVL C01677 V=800.0 PL=0
MOVL C01678 V=800.0 PL=0
MOVL C01679 V=800.0 PL=0
MOVL C01680 V=800.0 PL=0
MOVL C01681 V=800.0 PL=0
MOVL C01682 V=800.0 PL=0
MOVL C01683 V=800.0 PL=0
MOVL C01684 V=800.0 PL=0
MOVL C01685 V=800.0 PL=0
MOVL C01686 V=800.0 PL=0
MOVL C01687 V=800.0 PL=0
MOVL C01688 V=800.0 PL=0
MOVL C01689 V=800.0 PL=0
MOVL C01690 V=800.0 PL=0
MOVL C01691 V=800.0 PL=0
MOVL C01692 V=800.0 PL=0
MOVL C01693 V=800.0 PL=0
MOVL C01694 V=800.0 PL=0
MOVL C01695 V=800.0 PL=0
MOVL C01696 V=800.0 PL=0
MOVL C01697 V=800.0 PL=0
MOVL C01698 V=800.0 PL=0
MOVL C01699 V=800.0 PL=0
MOVL C01700 V=800.0 PL=0
MOVL C01701 V=800.0 PL=0
MOVL C01702 V=800.0 PL=0
MOVL C01703 V=800.0 PL=0
MOVL C01704 V=800.0 PL=0
MOVL C01705 V=800.0 PL=0
MOVL C01706 V=800.0 PL=0
MOVL C01707 V=800.0 PL=0
MOVL C01708 V=800.0 PL=0
MOVL C01709 V=800.0 PL=0
MOVL C01710 V=800.0 PL=0
MOVL C01711 V=800.0 PL=0
MOVL C01712 V=800.0 PL=0
MOVL C01713 V=800.0 PL=0
MOVL C01714 V=800.0 PL=0
MOVL C01715 V=800.0 PL=0
MOVL C01716 V=800.0 PL=0
MOVL C01717 V=800.0 PL=0
MOVL C01718 V=800.0 PL=0
MOVL C01719 V=800.0 PL=0
MOVL C01720 V=800.0 PL=0
MOVL C01721 V=800.0 PL=0
MOVL C01722 V=800.0 PL=0
MOVL C01723 V=800.0 PL=0
MOVL C01724 V=800.0 PL=0
MOVL C01725 V=800.0 PL=0
MOVL C01726 V=800.0 PL=0
MOVL C01727 V=800.0 PL=0
MOVL C01728 V=800.0 PL=0
MOVL C01729 V=800.0 PL=0
MOVL C01730 V=800.0 PL=0
MOVL C01731 V=800.0 PL=0
MOVL C01732 V=800.0 PL=0
MOVL C01733 V=800.0 PL=0
MOVL C01734 V=800.0 PL=0
MOVL C01735 V=800.0 PL=0
MOVL C01736 V=800.0 PL=0
MOVL C01737 V=800.0 PL=0
MOVL C01738 V=800.0 PL=0
MOVL C01739 V=800.0 PL=0
MOVL C01740 V=800.0 PL=0
MOVL C01741 V=800.0 PL=0
MOVL C01742 V=800.0 PL=0
MOVL C01743 V=800.0 PL=0
MOVL C01744 V=800.0 PL=0
MOVL C01745 V=800.0 PL=0
MOVL C01746 V=800.0 PL=0
MOVL C01747 V=800.0 PL=0
MOVL C01748 V=800.0 PL=0
MOVL C01749 V=800.0 PL=0
MOVL C01750 V=800.0 PL=0
MOVL C01751 V=800.0 PL=0
MOVL C01752 V=800.0 PL=0
MOVL C01753 V=800.0 PL=0
MOVL C01754 V=800.0 PL=0
MOVL C01755 V=800.0 PL=0
MOVL C01756 V=800.0 PL=0
MOVL C01757 V=800.0 PL=0
MOVL C01758 V=800.0 PL=0
MOVL C01759 V=800.0 PL=0
MOVL C01760 V=800.0 PL=0
MOVL C01761 V=800.0 PL=0
MOVL C01762 V=800.0 PL=0
MOVL C01763 V=800.0 PL=0
MOVL C01764 V=800.0 PL=0
MOVL C01765 V=800.0 PL=0
MOVL C01766 V=800.0 PL=0
MOVL C01767 V=800.0 PL=0
MOVL C01768 V=800.0 PL=0
MOVL C01769 V=800.0 PL=0
MOVL C01770 V=800.0 PL=0
MOVL C01771 V=800.0 PL=0
MOVL C01772 V=800.0 PL=0
MOVL C01773 V=800.0 PL=0
MOVL C01774 V=800.0 PL=0
MOVL C01775 V=800.0 PL=0
MOVL C01776 V=800.0 PL=0
MOVL C01777 V=800.0 PL=0
MOVL C01778 V=800.0 PL=0
MOVL C01779 V=800.0 PL=0
MOVL C01780 V=800.0 PL=0
MOVL C01781 V=800.0 PL=0
MOVL C01782 V=800.0 PL=0
MOVL C01783 V=800.0 PL=0
MOVL C01784 V=800.0 PL=0
MOVL C01785 V=800.0 PL=0
MOVL C01786 V=800.0 PL=0
MOVL C01787 V=800.0 PL=0
MOVL C01788 V=800.0 PL=0
MOVL C01789 V=800.0 PL=0
MOVL C01790 V=800.0 PL=0
MOVL C01791 V=800.0 PL=0
MOVL C01792 V=800.0 PL=0
MOVL C01793 V=800.0 PL=0
MOVL C01794 V=800.0 PL=0
MOVL C01795 V=800.0 PL=0
MOVL C01796 V=800.0 PL=0
MOVL C01797 V=800.0 PL=0
MOVL C01798 V=800.0 PL=0
MOVL C01799 V=800.0 PL=0
MOVL C01800 V=800.0 PL=0
MOVL C01801 V=800.0 PL=0
MOVL C01802 V=800.0 PL=0
MOVL C01803 V=800.0 PL=0
MOVL C01804 V=800.0 PL=0
MOVL C01805 V=800.0 PL=0
MOVL C01806 V=800.0 PL=0
MOVL C01807 V=800.0 PL=0
MOVL C01808 V=800.0 PL=0
MOVL C01809 V=800.0 PL=0
MOVL C01810 V=800.0 PL=0
MOVL C01811 V=800.0 PL=0
MOVL C01812 V=800.0 PL=0
MOVL C01813 V=800.0 PL=0
MOVL C01814 V=800.0 PL=0
MOVL C01815 V=800.0 PL=0
MOVL C01816 V=800.0 PL=0
MOVL C01817 V=800.0 PL=0
MOVL C01818 V=800.0 PL=0
MOVL C01819 V=800.0 PL=0
MOVL C01820 V=800.0 PL=0
MOVL C01821 V=800.0 PL=0
MOVL C01822 V=800.0 PL=0
MOVL C01823 V=800.0 PL=0
MOVL C01824 V=800.0 PL=0
MOVL C01825 V=800.0 PL=0
MOVL C01826 V=800.0 PL=0
MOVL C01827 V=800.0 PL=0
MOVL C01828 V=800.0 PL=0
MOVL C01829 V=800.0 PL=0
MOVL C01830 V=800.0 PL=0
MOVL C01831 V=800.0 PL=0
MOVL C01832 V=800.0 PL=0
MOVL C01833 V=800.0 PL=0
MOVL C01834 V=800.0 PL=0
MOVL C01835 V=800.0 PL=0
MOVL C01836 V=800.0 PL=0
MOVL C01837 V=800.0 PL=0
MOVL C01838 V=800.0 PL=0
MOVL C01839 V=800.0 PL=0
MOVL C01840 V=800.0 PL=0
MOVL C01841 V=800.0 PL=0
MOVL C01842 V=800.0 PL=0
MOVL C01843 V=800.0 PL=0
MOVL C01844 V=800.0 PL=0
MOVL C01845 V=800.0 PL=0
MOVL C01846 V=800.0 PL=0
MOVL C01847 V=800.0 PL=0
MOVL C01848 V=800.0 PL=0
MOVL C01849 V=800.0 PL=0
MOVL C01850 V=800.0 PL=0
MOVL C01851 V=800.0 PL=0
MOVL C01852 V=800.0 PL=0
MOVL C01853 V=800.0 PL=0
MOVL C01854 V=800.0 PL=0
MOVL C01855 V=800.0 PL=0
MOVL C01856 V=800.0 PL=0
MOVL C01857 V=800.0 PL=0
MOVL C01858 V=800.0 PL=0
MOVL C01859 V=800.0 PL=0
MOVL C01860 V=800.0 PL=0
MOVL C01861 V=800.0 PL=0
MOVL C01862 V=800.0 PL=0
MOVL C01863 V=800.0 PL=0
MOVL C01864 V=800.0 PL=0
MOVL C01865 V=800.0 PL=0
MOVL C01866 V=800.0 PL=0
MOVL C01867 V=800.0 PL=0
MOVL C01868 V=800.0 PL=0
MOVL C01869 V=800.0 PL=0
MOVL C01870 V=800.0 PL=0
MOVL C01871 V=800.0 PL=0
MOVL C01872 V=800.0 PL=0
MOVL C01873 V=800.0 PL=0
MOVL C01874 V=800.0 PL=0
MOVL C01875 V=800.0 PL=0
MOVL C01876 V=800.0 PL=0
MOVL C01877 V=800.0 PL=0
MOVL C01878 V=800.0 PL=0
MOVL C01879 V=800.0 PL=0
MOVL C01880 V=800.0 PL=0
MOVL C01881 V=800.0 PL=0
MOVL C01882 V=800.0 PL=0
MOVL C01883 V=800.0 PL=0
MOVL C01884 V=800.0 PL=0
MOVL C01885 V=800.0 PL=0
MOVL C01886 V=800.0 PL=0
MOVL C01887 V=800.0 PL=0
MOVL C01888 V=800.0 PL=0
MOVL C01889 V=800.0 PL=0
MOVL C01890 V=800.0 PL=0
MOVL C01891 V=800.0 PL=0
MOVL C01892 V=800.0 PL=0
MOVL C01893 V=800.0 PL=0
MOVL C01894 V=800.0 PL=0
MOVL C01895 V=800.0 PL=0
MOVL C01896 V=800.0 PL=0
MOVL C01897 V=800.0 PL=0
MOVL C01898 V=800.0 PL=0
MOVL C01899 V=800.0 PL=0
MOVL C01900 V=800.0 PL=0
MOVL C01901 V=800.0 PL=0
MOVL C01902 V=800.0 PL=0
MOVL C01903 V=800.0 PL=0
MOVL C01904 V=800.0 PL=0
MOVL C01905 V=800.0 PL=0
MOVL C01906 V=800.0 PL=0
MOVL C01907 V=800.0 PL=0
MOVL C01908 V=800.0 PL=0
MOVL C01909 V=800.0 PL=0
MOVL C01910 V=800.0 PL=0
MOVL C01911 V=800.0 PL=0
MOVL C01912 V=800.0 PL=0
MOVL C01913 V=800.0 PL=0
MOVL C01914 V=800.0 PL=0
MOVL C01915 V=800.0 PL=0
MOVL C01916 V=800.0 PL=0
MOVL C01917 V=800.0 PL=0
MOVL C01918 V=800.0 PL=0
MOVL C01919 V=800.0 PL=0
MOVL C01920 V=800.0 PL=0
MOVL C01921 V=800.0 PL=0
MOVL C01922 V=800.0 PL=0
MOVL C01923 V=800.0 PL=0
MOVL C01924 V=800.0 PL=0
MOVL C01925 V=800.0 PL=0
MOVL C01926 V=800.0 PL=0
MOVL C01927 V=800.0 PL=0
MOVL C01928 V=800.0 PL=0
MOVL C01929 V=800.0 PL=0
MOVL C01930 V=800.0 PL=0
MOVL C01931 V=800.0 PL=0
MOVL C01932 V=800.0 PL=0
MOVL C01933 V=800.0 PL=0
MOVL C01934 V=800.0 PL=0
MOVL C01935 V=800.0 PL=0
MOVL C01936 V=800.0 PL=0
MOVL C01937 V=800.0 PL=0
MOVL C01938 V=800.0 PL=0
MOVL C01939 V=800.0 PL=0
MOVL C01940 V=800.0 PL=0
MOVL C01941 V=800.0 PL=0
MOVL C01942 V=800.0 PL=0
MOVL C01943 V=800.0 PL=0
MOVL C01944 V=800.0 PL=0
MOVL C01945 V=800.0 PL=0
MOVL C01946 V=800.0 PL=0
MOVL C01947 V=800.0 PL=0
MOVL C01948 V=800.0 PL=0
MOVL C01949 V=800.0 PL=0
MOVL C01950 V=800.0 PL=0
MOVL C01951 V=800.0 PL=0
MOVL C01952 V=800.0 PL=0
MOVL C01953 V=800.0 PL=0
MOVL C01954 V=800.0 PL=0
MOVL C01955 V=800.0 PL=0
MOVL C01956 V=800.0 PL=0
MOVL C01957 V=800.0 PL=0
MOVL C01958 V=800.0 PL=0
MOVL C01959 V=800.0 PL=0
MOVL C01960 V=800.0 PL=0
MOVL C01961 V=800.0 PL=0
MOVL C01962 V=800.0 PL=0
MOVL C01963 V=800.0 PL=0
MOVL C01964 V=800.0 PL=0
MOVL C01965 V=800.0 PL=0
MOVL C01966 V=800.0 PL=0
MOVL C01967 V=800.0 PL=0
MOVL C01968 V=800.0 PL=0
MOVL C01969 V=800.0 PL=0
MOVL C01970 V=800.0 PL=0
